Universal Robots PolyScope program: 2024dragon.urp

Program 2024dragon (installation=default directory=/programs createdIn=5.11.9.1010452 lastSavedIn=5.11.9.1010452 robotSerialNumber=20225200364)
Calibrated DH parameters: a=[0.00002, -0.569483, -0.54992, -0.00001, -0.000036, 0]; d=[0.180894, -146.691669, 192.918669, -46.053088, 0.119778, 0.115602]; alpha=[1.571425, -0.001534, 0.003359, 1.568739, -1.571477, 0]; deltaTheta=[0, 0.376258, -0.101074, -0.275185, -0.000002, 0]
Robot Program (runOnlyOnce=true)
  Script file /programs/usbdisk/new-robot/2024Dragon.script
    | def Machining1():
    |   # Default parameters:
    |   global speed_ms = 0.3
    |   global speed_rads = 0.75
    |   global accel_mss = 3
    |   global accel_radss = 1.2
    |   global blend_radius_m = 0.001
    | 
    |   # Add subprograms here
    |   # Start of main program
    |   # Program generated by RoboDK v5.6.5 for UR10e on 10/01/2024 16:23:47
    |   # Using nominal kinematics.
    |   blend_radius_m = 0.001
    |   speed_ms = 1.000
    |   # set_reference(p[0.335000, -0.152000, 0.002000, 0.000000, 0.000000, 0.000000])
    |   set_tcp(p[0.000000, 0.000000, 0.252000, 0.000000, 0.000000, 0.000000])
    |   # Show Tool
    |   movej([0.067194, -1.074636, -2.586948, -1.050805, 1.570796, 1.637990],accel_radss,speed_rads,0,blend_radius_m)
    |   movel([0.067194, -1.074636, -2.586948, -1.050805, 1.570796, 1.637990],accel_mss,speed_ms,0,blend_radius_m)
    |   # Splitting Linear movement in 32 (instruction 7: MoveL 3)
    |   movel([0.067194, -1.076085, -2.588243, -1.048061, 1.570796, 1.637990],accel_mss,speed_ms,0,blend_radius_m)
    |   movel([0.067194, -1.077544, -2.589536, -1.045309, 1.570796, 1.637990],accel_mss,speed_ms,0,blend_radius_m)
    |   movel([0.067194, -1.079013, -2.590827, -1.042549, 1.570796, 1.637990],accel_mss,speed_ms,0,blend_radius_m)
    |   movel([0.067194, -1.080492, -2.592116, -1.039781, 1.570796, 1.637990],accel_mss,speed_ms,0,blend_radius_m)
    |   movel([0.067194, -1.081981, -2.593403, -1.037005, 1.570796, 1.637990],accel_mss,speed_ms,0,blend_radius_m)
    |   movel([0.067194, -1.083480, -2.594688, -1.034221, 1.570796, 1.637990],accel_mss,speed_ms,0,blend_radius_m)
    |   movel([0.067194, -1.084989, -2.595971, -1.031429, 1.570796, 1.637990],accel_mss,speed_ms,0,blend_radius_m)
    |   movel([0.067194, -1.086509, -2.597251, -1.028629, 1.570796, 1.637990],accel_mss,speed_ms,0,blend_radius_m)
    |   movel([0.067194, -1.088039, -2.598529, -1.025821, 1.570796, 1.637990],accel_mss,speed_ms,0,blend_radius_m)
    |   movel([0.067194, -1.089579, -2.599806, -1.023004, 1.570796, 1.637990],accel_mss,speed_ms,0,blend_radius_m)
    |   movel([0.067194, -1.091130, -2.601080, -1.020179, 1.570796, 1.637990],accel_mss,speed_ms,0,blend_radius_m)
    |   movel([0.067194, -1.092691, -2.602351, -1.017346, 1.570796, 1.637990],accel_mss,speed_ms,0,blend_radius_m)
    |   movel([0.067194, -1.094263, -2.603621, -1.014505, 1.570796, 1.637990],accel_mss,speed_ms,0,blend_radius_m)
    |   movel([0.067194, -1.095846, -2.604888, -1.011655, 1.570796, 1.637990],accel_mss,speed_ms,0,blend_radius_m)
    |   movel([0.067194, -1.097439, -2.606154, -1.008797, 1.570796, 1.637990],accel_mss,speed_ms,0,blend_radius_m)
    |   movel([0.067194, -1.099042, -2.607417, -1.005930, 1.570796, 1.637990],accel_mss,speed_ms,0,blend_radius_m)
    |   movel([0.067194, -1.100657, -2.608677, -1.003055, 1.570796, 1.637990],accel_mss,speed_ms,0,blend_radius_m)
    |   movel([0.067194, -1.102282, -2.609936, -1.000171, 1.570796, 1.637990],accel_mss,speed_ms,0,blend_radius_m)
    |   movel([0.067194, -1.103918, -2.611192, -0.997279, 1.570796, 1.637990],accel_mss,speed_ms,0,blend_radius_m)
    |   movel([0.067194, -1.105565, -2.612446, -0.994378, 1.570796, 1.637990],accel_mss,speed_ms,0,blend_radius_m)
    |   movel([0.067194, -1.107223, -2.613698, -0.991469, 1.570796, 1.637990],accel_mss,speed_ms,0,blend_radius_m)
    |   movel([0.067194, -1.108891, -2.614947, -0.988551, 1.570796, 1.637990],accel_mss,speed_ms,0,blend_radius_m)
    |   movel([0.067194, -1.110571, -2.616194, -0.985624, 1.570796, 1.637990],accel_mss,speed_ms,0,blend_radius_m)
    |   movel([0.067194, -1.112262, -2.617439, -0.982688, 1.570796, 1.637990],accel_mss,speed_ms,0,blend_radius_m)
    |   movel([0.067194, -1.113964, -2.618681, -0.979744, 1.570796, 1.637990],accel_mss,speed_ms,0,blend_radius_m)
    |   movel([0.067194, -1.115677, -2.619921, -0.976791, 1.570796, 1.637990],accel_mss,speed_ms,0,blend_radius_m)
    |   movel([0.067194, -1.117402, -2.621159, -0.973829, 1.570796, 1.637990],accel_mss,speed_ms,0,blend_radius_m)
    |   movel([0.067194, -1.119137, -2.622394, -0.970858, 1.570796, 1.637990],accel_mss,speed_ms,0,blend_radius_m)
    |   movel([0.067194, -1.120884, -2.623627, -0.967878, 1.570796, 1.637990],accel_mss,speed_ms,0,blend_radius_m)
    |   movel([0.067194, -1.122643, -2.624857, -0.964889, 1.570796, 1.637990],accel_mss,speed_ms,0,blend_radius_m)
    |   movel([0.067194, -1.124413, -2.626085, -0.961891, 1.570796, 1.637990],accel_mss,speed_ms,0,blend_radius_m)
    |   movel([0.067194, -1.126194, -2.627311, -0.958884, 1.570796, 1.637990],accel_mss,speed_ms,0,blend_radius_m)
    |   movel([0.067194, -1.126194, -2.627311, -0.958884, 1.570796, 1.637990],accel_mss,speed_ms,0,blend_radius_m)
    |   speed_ms = 1.000
    |   movel([0.067194, -1.126194, -2.627311, -0.958884, 1.570796, 1.637990],accel_mss,speed_ms,0,blend_radius_m)
    |   movel([0.067194, -1.126194, -2.627311, -0.958884, 1.570796, 1.637990],accel_mss,speed_ms,0,blend_radius_m)
    |   movel([0.067194, -1.126194, -2.627311, -0.958884, 1.570796, 1.637990],accel_mss,speed_ms,0,blend_radius_m)
    |   speed_ms = 0.005
    |   # Splitting Linear movement in 22 (instruction 14: MoveL 8)
    |   movel([0.067194, -1.124466, -2.626123, -0.961800, 1.570796, 1.637990],accel_mss,speed_ms,0,blend_radius_m)
    |   movel([0.067194, -1.122750, -2.624932, -0.964708, 1.570796, 1.637990],accel_mss,speed_ms,0,blend_radius_m)
    |   movel([0.067194, -1.121044, -2.623739, -0.967606, 1.570796, 1.637990],accel_mss,speed_ms,0,blend_radius_m)
    |   movel([0.067194, -1.119348, -2.622544, -0.970497, 1.570796, 1.637990],accel_mss,speed_ms,0,blend_radius_m)
    |   movel([0.067194, -1.117664, -2.621346, -0.973379, 1.570796, 1.637990],accel_mss,speed_ms,0,blend_radius_m)
    |   movel([0.067194, -1.115990, -2.620146, -0.976253, 1.570796, 1.637990],accel_mss,speed_ms,0,blend_radius_m)
    |   movel([0.067194, -1.114326, -2.618944, -0.979118, 1.570796, 1.637990],accel_mss,speed_ms,0,blend_radius_m)
    |   movel([0.067194, -1.112674, -2.617740, -0.981975, 1.570796, 1.637990],accel_mss,speed_ms,0,blend_radius_m)
    |   movel([0.067194, -1.111031, -2.616534, -0.984824, 1.570796, 1.637990],accel_mss,speed_ms,0,blend_radius_m)
    |   movel([0.067194, -1.109399, -2.615325, -0.987665, 1.570796, 1.637990],accel_mss,speed_ms,0,blend_radius_m)
    |   movel([0.067194, -1.107778, -2.614114, -0.990497, 1.570796, 1.637990],accel_mss,speed_ms,0,blend_radius_m)
    |   movel([0.067194, -1.106166, -2.612901, -0.993321, 1.570796, 1.637990],accel_mss,speed_ms,0,blend_radius_m)
    |   movel([0.067194, -1.104565, -2.611686, -0.996137, 1.570796, 1.637990],accel_mss,speed_ms,0,blend_radius_m)
    |   movel([0.067194, -1.102975, -2.610469, -0.998945, 1.570796, 1.637990],accel_mss,speed_ms,0,blend_radius_m)
    |   movel([0.067194, -1.101394, -2.609250, -1.001745, 1.570796, 1.637990],accel_mss,speed_ms,0,blend_radius_m)
    |   movel([0.067194, -1.099824, -2.608028, -1.004537, 1.570796, 1.637990],accel_mss,speed_ms,0,blend_radius_m)
    |   movel([0.067194, -1.098263, -2.606805, -1.007321, 1.570796, 1.637990],accel_mss,speed_ms,0,blend_radius_m)
    |   movel([0.067194, -1.096713, -2.605579, -1.010097, 1.570796, 1.637990],accel_mss,speed_ms,0,blend_radius_m)
    |   movel([0.067194, -1.095173, -2.604351, -1.012865, 1.570796, 1.637990],accel_mss,speed_ms,0,blend_radius_m)
    |   movel([0.067194, -1.093643, -2.603121, -1.015625, 1.570796, 1.637990],accel_mss,speed_ms,0,blend_radius_m)
    |   movel([0.067194, -1.092123, -2.601889, -1.018377, 1.570796, 1.637990],accel_mss,speed_ms,0,blend_radius_m)
    |   movel([0.067194, -1.090612, -2.600655, -1.021122, 1.570796, 1.637990],accel_mss,speed_ms,0,blend_radius_m)
    |   speed_ms = 1.000
    |   # Splitting Linear movement in 22 (instruction 16: MoveL 9)
    |   movel([0.067194, -1.092123, -2.601889, -1.018377, 1.570796, 1.637990],accel_mss,speed_ms,0,blend_radius_m)
    |   movel([0.067194, -1.093643, -2.603121, -1.015625, 1.570796, 1.637990],accel_mss,speed_ms,0,blend_radius_m)
    |   movel([0.067194, -1.095173, -2.604351, -1.012865, 1.570796, 1.637990],accel_mss,speed_ms,0,blend_radius_m)
    |   movel([0.067194, -1.096713, -2.605579, -1.010097, 1.570796, 1.637990],accel_mss,speed_ms,0,blend_radius_m)
    |   movel([0.067194, -1.098263, -2.606805, -1.007321, 1.570796, 1.637990],accel_mss,speed_ms,0,blend_radius_m)
    |   movel([0.067194, -1.099824, -2.608028, -1.004537, 1.570796, 1.637990],accel_mss,speed_ms,0,blend_radius_m)
    |   movel([0.067194, -1.101394, -2.609250, -1.001745, 1.570796, 1.637990],accel_mss,speed_ms,0,blend_radius_m)
    |   movel([0.067194, -1.102975, -2.610469, -0.998945, 1.570796, 1.637990],accel_mss,speed_ms,0,blend_radius_m)
    |   movel([0.067194, -1.104565, -2.611686, -0.996137, 1.570796, 1.637990],accel_mss,speed_ms,0,blend_radius_m)
    |   movel([0.067194, -1.106166, -2.612901, -0.993321, 1.570796, 1.637990],accel_mss,speed_ms,0,blend_radius_m)
    |   movel([0.067194, -1.107778, -2.614114, -0.990497, 1.570796, 1.637990],accel_mss,speed_ms,0,blend_radius_m)
    |   movel([0.067194, -1.109399, -2.615325, -0.987665, 1.570796, 1.637990],accel_mss,speed_ms,0,blend_radius_m)
    |   movel([0.067194, -1.111031, -2.616534, -0.984824, 1.570796, 1.637990],accel_mss,speed_ms,0,blend_radius_m)
    |   movel([0.067194, -1.112674, -2.617740, -0.981975, 1.570796, 1.637990],accel_mss,speed_ms,0,blend_radius_m)
    |   movel([0.067194, -1.114326, -2.618944, -0.979118, 1.570796, 1.637990],accel_mss,speed_ms,0,blend_radius_m)
    |   movel([0.067194, -1.115990, -2.620146, -0.976253, 1.570796, 1.637990],accel_mss,speed_ms,0,blend_radius_m)
    |   movel([0.067194, -1.117664, -2.621346, -0.973379, 1.570796, 1.637990],accel_mss,speed_ms,0,blend_radius_m)
    |   movel([0.067194, -1.119348, -2.622544, -0.970497, 1.570796, 1.637990],accel_mss,speed_ms,0,blend_radius_m)
    |   movel([0.067194, -1.121044, -2.623739, -0.967606, 1.570796, 1.637990],accel_mss,speed_ms,0,blend_radius_m)
    |   movel([0.067194, -1.122750, -2.624932, -0.964708, 1.570796, 1.637990],accel_mss,speed_ms,0,blend_radius_m)
    |   movel([0.067194, -1.124466, -2.626123, -0.961800, 1.570796, 1.637990],accel_mss,speed_ms,0,blend_radius_m)
    |   movel([0.067194, -1.126194, -2.627311, -0.958884, 1.570796, 1.637990],accel_mss,speed_ms,0,blend_radius_m)
    |   speed_ms = 0.040
    |   movel([0.067194, -1.126194, -2.627311, -0.958884, 1.570796, 1.637990],accel_mss,speed_ms,0,blend_radius_m)
    |   speed_ms = 1.000
    |   movel([0.067194, -1.126194, -2.627311, -0.958884, 1.570796, 1.637990],accel_mss,speed_ms,0,blend_radius_m)
    |   # Splitting Linear movement in 38 (instruction 21: MoveL 12)
    |   movel([0.069828, -1.126252, -2.627286, -0.958852, 1.570796, 1.640625],accel_mss,speed_ms,0,blend_radius_m)
    |   movel([0.072458, -1.126317, -2.627257, -0.958815, 1.570796, 1.643255],accel_mss,speed_ms,0,blend_radius_m)
    |   movel([0.075084, -1.126391, -2.627225, -0.958773, 1.570796, 1.645881],accel_mss,speed_ms,0,blend_radius_m)
    |   movel([0.077706, -1.126473, -2.627189, -0.958727, 1.570796, 1.648503],accel_mss,speed_ms,0,blend_radius_m)
    |   movel([0.080324, -1.126562, -2.627150, -0.958677, 1.570796, 1.651120],accel_mss,speed_ms,0,blend_radius_m)
    |   movel([0.082938, -1.126660, -2.627107, -0.958622, 1.570796, 1.653734],accel_mss,speed_ms,0,blend_radius_m)
    |   movel([0.085547, -1.126766, -2.627061, -0.958562, 1.570796, 1.656343],accel_mss,speed_ms,0,blend_radius_m)
    |   movel([0.088152, -1.126880, -2.627011, -0.958498, 1.570796, 1.658948],accel_mss,speed_ms,0,blend_radius_m)
    |   movel([0.090752, -1.127001, -2.626958, -0.958430, 1.570796, 1.661549],accel_mss,speed_ms,0,blend_radius_m)
    |   movel([0.093349, -1.127131, -2.626901, -0.958357, 1.570796, 1.664145],accel_mss,speed_ms,0,blend_radius_m)
    |   movel([0.095940, -1.127269, -2.626841, -0.958279, 1.570796, 1.666737],accel_mss,speed_ms,0,blend_radius_m)
    |   movel([0.098528, -1.127415, -2.626777, -0.958197, 1.570796, 1.669324],accel_mss,speed_ms,0,blend_radius_m)
    |   movel([0.101111, -1.127568, -2.626710, -0.958111, 1.570796, 1.671907],accel_mss,speed_ms,0,blend_radius_m)
    |   movel([0.103689, -1.127730, -2.626639, -0.958020, 1.570796, 1.674485],accel_mss,speed_ms,0,blend_radius_m)
    |   movel([0.106263, -1.127899, -2.626565, -0.957925, 1.570796, 1.677059],accel_mss,speed_ms,0,blend_radius_m)
    |   movel([0.108832, -1.128077, -2.626487, -0.957825, 1.570796, 1.679629],accel_mss,speed_ms,0,blend_radius_m)
    |   movel([0.111397, -1.128262, -2.626406, -0.957721, 1.570796, 1.682193],accel_mss,speed_ms,0,blend_radius_m)
    |   movel([0.113957, -1.128456, -2.626321, -0.957612, 1.570796, 1.684754],accel_mss,speed_ms,0,blend_radius_m)
    |   movel([0.116513, -1.128657, -2.626233, -0.957499, 1.570796, 1.687309],accel_mss,speed_ms,0,blend_radius_m)
    |   movel([0.119064, -1.128866, -2.626141, -0.957382, 1.570796, 1.689860],accel_mss,speed_ms,0,blend_radius_m)
    |   movel([0.121610, -1.129083, -2.626045, -0.957260, 1.570796, 1.692406],accel_mss,speed_ms,0,blend_radius_m)
    |   movel([0.124151, -1.129308, -2.625947, -0.957134, 1.570796, 1.694947],accel_mss,speed_ms,0,blend_radius_m)
    |   movel([0.126687, -1.129541, -2.625844, -0.957004, 1.570796, 1.697484],accel_mss,speed_ms,0,blend_radius_m)
    |   movel([0.129219, -1.129781, -2.625738, -0.956869, 1.570796, 1.700016],accel_mss,speed_ms,0,blend_radius_m)
    |   movel([0.131746, -1.130030, -2.625629, -0.956730, 1.570796, 1.702542],accel_mss,speed_ms,0,blend_radius_m)
    |   movel([0.134268, -1.130286, -2.625516, -0.956587, 1.570796, 1.705065],accel_mss,speed_ms,0,blend_radius_m)
    |   movel([0.136785, -1.130550, -2.625400, -0.956439, 1.570796, 1.707582],accel_mss,speed_ms,0,blend_radius_m)
    |   movel([0.139298, -1.130822, -2.625280, -0.956287, 1.570796, 1.710094],accel_mss,speed_ms,0,blend_radius_m)
    |   movel([0.141805, -1.131102, -2.625156, -0.956131, 1.570796, 1.712601],accel_mss,speed_ms,0,blend_radius_m)
    |   movel([0.144307, -1.131389, -2.625030, -0.955970, 1.570796, 1.715104],accel_mss,speed_ms,0,blend_radius_m)
    |   movel([0.146805, -1.131684, -2.624899, -0.955805, 1.570796, 1.717601],accel_mss,speed_ms,0,blend_radius_m)
    |   movel([0.149297, -1.131987, -2.624765, -0.955636, 1.570796, 1.720093],accel_mss,speed_ms,0,blend_radius_m)
    |   movel([0.151784, -1.132298, -2.624628, -0.955463, 1.570796, 1.722581],accel_mss,speed_ms,0,blend_radius_m)
    |   movel([0.154267, -1.132616, -2.624487, -0.955286, 1.570796, 1.725063],accel_mss,speed_ms,0,blend_radius_m)
    |   movel([0.156744, -1.132942, -2.624343, -0.955104, 1.570796, 1.727540],accel_mss,speed_ms,0,blend_radius_m)
    |   movel([0.159216, -1.133276, -2.624195, -0.954918, 1.570796, 1.730012],accel_mss,speed_ms,0,blend_radius_m)
    |   movel([0.161683, -1.133617, -2.624043, -0.954728, 1.570796, 1.732479],accel_mss,speed_ms,0,blend_radius_m)
    |   movel([0.164144, -1.133966, -2.623888, -0.954534, 1.570796, 1.734941],accel_mss,speed_ms,0,blend_radius_m)
    |   speed_ms = 0.005
    |   # Splitting Linear movement in 22 (instruction 23: MoveL 13)
    |   movel([0.164144, -1.135705, -2.625067, -0.951617, 1.570796, 1.734941],accel_mss,speed_ms,0,blend_radius_m)
    |   movel([0.164144, -1.137454, -2.626244, -0.948691, 1.570796, 1.734941],accel_mss,speed_ms,0,blend_radius_m)
    |   movel([0.164144, -1.139214, -2.627418, -0.945757, 1.570796, 1.734941],accel_mss,speed_ms,0,blend_radius_m)
    |   movel([0.164144, -1.140985, -2.628590, -0.942814, 1.570796, 1.734941],accel_mss,speed_ms,0,blend_radius_m)
    |   movel([0.164144, -1.142767, -2.629760, -0.939862, 1.570796, 1.734941],accel_mss,speed_ms,0,blend_radius_m)
    |   movel([0.164144, -1.144560, -2.630927, -0.936902, 1.570796, 1.734941],accel_mss,speed_ms,0,blend_radius_m)
    |   movel([0.164144, -1.146364, -2.632091, -0.933934, 1.570796, 1.734941],accel_mss,speed_ms,0,blend_radius_m)
    |   movel([0.164144, -1.148179, -2.633254, -0.930957, 1.570796, 1.734941],accel_mss,speed_ms,0,blend_radius_m)
    |   movel([0.164144, -1.150005, -2.634414, -0.927971, 1.570796, 1.734941],accel_mss,speed_ms,0,blend_radius_m)
    |   movel([0.164144, -1.151842, -2.635571, -0.924976, 1.570796, 1.734941],accel_mss,speed_ms,0,blend_radius_m)
    |   movel([0.164144, -1.153690, -2.636726, -0.921973, 1.570796, 1.734941],accel_mss,speed_ms,0,blend_radius_m)
    |   movel([0.164144, -1.155550, -2.637879, -0.918961, 1.570796, 1.734941],accel_mss,speed_ms,0,blend_radius_m)
    |   movel([0.164144, -1.157420, -2.639029, -0.915940, 1.570796, 1.734941],accel_mss,speed_ms,0,blend_radius_m)
    |   movel([0.164144, -1.159302, -2.640176, -0.912911, 1.570796, 1.734941],accel_mss,speed_ms,0,blend_radius_m)
    |   movel([0.164144, -1.161196, -2.641321, -0.909872, 1.570796, 1.734941],accel_mss,speed_ms,0,blend_radius_m)
    |   movel([0.164144, -1.163101, -2.642463, -0.906825, 1.570796, 1.734941],accel_mss,speed_ms,0,blend_radius_m)
    |   movel([0.164144, -1.165017, -2.643603, -0.903769, 1.570796, 1.734941],accel_mss,speed_ms,0,blend_radius_m)
    |   movel([0.164144, -1.166945, -2.644741, -0.900704, 1.570796, 1.734941],accel_mss,speed_ms,0,blend_radius_m)
    |   movel([0.164144, -1.168884, -2.645876, -0.897629, 1.570796, 1.734941],accel_mss,speed_ms,0,blend_radius_m)
    |   movel([0.164144, -1.170835, -2.647008, -0.894546, 1.570796, 1.734941],accel_mss,speed_ms,0,blend_radius_m)
    |   movel([0.164144, -1.172797, -2.648137, -0.891454, 1.570796, 1.734941],accel_mss,speed_ms,0,blend_radius_m)
    |   movel([0.164144, -1.174772, -2.649264, -0.888353, 1.570796, 1.734941],accel_mss,speed_ms,0,blend_radius_m)
    |   speed_ms = 0.035
    |   movel([0.164993, -1.172613, -2.650270, -0.889506, 1.570796, 1.735790],accel_mss,speed_ms,0,blend_radius_m)
    |   movel([0.165155, -1.171113, -2.650966, -0.890310, 1.570796, 1.735952],accel_mss,speed_ms,0,blend_radius_m)
    |   movel([0.164874, -1.170165, -2.651404, -0.890819, 1.570796, 1.735671],accel_mss,speed_ms,0,blend_radius_m)
    |   movel([0.164399, -1.169671, -2.651633, -0.891085, 1.570796, 1.735195],accel_mss,speed_ms,0,blend_radius_m)
    |   movel([0.161880, -1.168870, -2.652002, -0.891517, 1.570796, 1.732676],accel_mss,speed_ms,0,blend_radius_m)
    |   movel([0.161427, -1.168227, -2.652299, -0.891864, 1.570796, 1.732224],accel_mss,speed_ms,0,blend_radius_m)
    |   movel([0.161378, -1.167640, -2.652568, -0.892180, 1.570796, 1.732174],accel_mss,speed_ms,0,blend_radius_m)
    |   movel([0.161619, -1.166900, -2.652908, -0.892581, 1.570796, 1.732416],accel_mss,speed_ms,0,blend_radius_m)
    |   movel([0.162186, -1.166146, -2.653254, -0.892989, 1.570796, 1.732982],accel_mss,speed_ms,0,blend_radius_m)
    |   movel([0.162955, -1.165553, -2.653526, -0.893311, 1.570796, 1.733751],accel_mss,speed_ms,0,blend_radius_m)
    |   movel([0.163842, -1.165169, -2.653701, -0.893519, 1.570796, 1.734638],accel_mss,speed_ms,0,blend_radius_m)
    |   movel([0.164754, -1.165038, -2.653761, -0.893590, 1.570796, 1.735550],accel_mss,speed_ms,0,blend_radius_m)
    |   movel([0.166318, -1.164944, -2.653804, -0.893641, 1.570796, 1.737114],accel_mss,speed_ms,0,blend_radius_m)
    |   movel([0.167392, -1.164661, -2.653933, -0.893795, 1.570796, 1.738188],accel_mss,speed_ms,0,blend_radius_m)
    |   movel([0.168112, -1.164264, -2.654114, -0.894010, 1.570796, 1.738908],accel_mss,speed_ms,0,blend_radius_m)
    |   movel([0.168622, -1.163824, -2.654315, -0.894250, 1.570796, 1.739418],accel_mss,speed_ms,0,blend_radius_m)
    |   movel([0.169089, -1.163137, -2.654628, -0.894624, 1.570796, 1.739886],accel_mss,speed_ms,0,blend_radius_m)
    |   movel([0.169480, -1.162013, -2.655138, -0.895237, 1.570796, 1.740276],accel_mss,speed_ms,0,blend_radius_m)
    |   movel([0.169481, -1.161424, -2.655406, -0.895560, 1.570796, 1.740277],accel_mss,speed_ms,0,blend_radius_m)
    |   movel([0.169274, -1.160885, -2.655650, -0.895854, 1.570796, 1.740071],accel_mss,speed_ms,0,blend_radius_m)
    |   movel([0.168785, -1.160454, -2.655845, -0.896090, 1.570796, 1.739581],accel_mss,speed_ms,0,blend_radius_m)
    |   movel([0.167958, -1.160181, -2.655968, -0.896240, 1.570796, 1.738755],accel_mss,speed_ms,0,blend_radius_m)
    |   speed_ms = 0.005
    |   # Splitting Linear movement in 6 (instruction 48: MoveL 36)
    |   movel([0.167958, -1.158728, -2.655131, -0.898529, 1.570796, 1.738755],accel_mss,speed_ms,0,blend_radius_m)
    |   movel([0.167958, -1.157282, -2.654293, -0.900814, 1.570796, 1.738755],accel_mss,speed_ms,0,blend_radius_m)
    |   movel([0.167958, -1.155842, -2.653454, -0.903093, 1.570796, 1.738755],accel_mss,speed_ms,0,blend_radius_m)
    |   movel([0.167958, -1.154408, -2.652613, -0.905368, 1.570796, 1.738755],accel_mss,speed_ms,0,blend_radius_m)
    |   movel([0.167958, -1.152981, -2.651771, -0.907637, 1.570796, 1.738755],accel_mss,speed_ms,0,blend_radius_m)
    |   movel([0.167958, -1.151560, -2.650928, -0.909901, 1.570796, 1.738755],accel_mss,speed_ms,0,blend_radius_m)
    |   speed_ms = 0.040
    |   # Splitting Linear movement in 4 (instruction 50: MoveL 37)
    |   movel([0.168272, -1.153369, -2.650117, -0.908903, 1.570796, 1.739068],accel_mss,speed_ms,0,blend_radius_m)
    |   movel([0.168584, -1.155175, -2.649304, -0.907909, 1.570796, 1.739381],accel_mss,speed_ms,0,blend_radius_m)
    |   movel([0.168895, -1.156978, -2.648490, -0.906921, 1.570796, 1.739692],accel_mss,speed_ms,0,blend_radius_m)
    |   movel([0.169205, -1.158777, -2.647674, -0.905937, 1.570796, 1.740001],accel_mss,speed_ms,0,blend_radius_m)
    |   speed_ms = 0.005
    |   # Splitting Linear movement in 6 (instruction 52: MoveL 38)
    |   movel([0.169205, -1.160197, -2.648513, -0.903680, 1.570796, 1.740001],accel_mss,speed_ms,0,blend_radius_m)
    |   movel([0.169205, -1.161622, -2.649350, -0.901417, 1.570796, 1.740001],accel_mss,speed_ms,0,blend_radius_m)
    |   movel([0.169205, -1.163054, -2.650186, -0.899149, 1.570796, 1.740001],accel_mss,speed_ms,0,blend_radius_m)
    |   movel([0.169205, -1.164492, -2.651020, -0.896877, 1.570796, 1.740001],accel_mss,speed_ms,0,blend_radius_m)
    |   movel([0.169205, -1.165937, -2.651853, -0.894599, 1.570796, 1.740001],accel_mss,speed_ms,0,blend_radius_m)
    |   movel([0.169205, -1.167388, -2.652684, -0.892317, 1.570796, 1.740001],accel_mss,speed_ms,0,blend_radius_m)
    |   speed_ms = 0.035
    |   movel([0.170114, -1.166953, -2.652884, -0.892552, 1.570796, 1.740910],accel_mss,speed_ms,0,blend_radius_m)
    |   movel([0.170952, -1.166789, -2.652959, -0.892641, 1.570796, 1.741748],accel_mss,speed_ms,0,blend_radius_m)
    |   movel([0.171650, -1.166893, -2.652911, -0.892584, 1.570796, 1.742446],accel_mss,speed_ms,0,blend_radius_m)
    |   movel([0.172147, -1.167265, -2.652741, -0.892383, 1.570796, 1.742943],accel_mss,speed_ms,0,blend_radius_m)
    |   movel([0.172364, -1.167756, -2.652515, -0.892118, 1.570796, 1.743160],accel_mss,speed_ms,0,blend_radius_m)
    |   movel([0.172398, -1.168357, -2.652239, -0.891793, 1.570796, 1.743194],accel_mss,speed_ms,0,blend_radius_m)
    |   movel([0.172257, -1.169008, -2.651939, -0.891442, 1.570796, 1.743053],accel_mss,speed_ms,0,blend_radius_m)
    |   movel([0.171937, -1.169655, -2.651640, -0.891094, 1.570796, 1.742733],accel_mss,speed_ms,0,blend_radius_m)
    |   movel([0.170592, -1.171154, -2.650947, -0.890288, 1.570796, 1.741389],accel_mss,speed_ms,0,blend_radius_m)
    |   movel([0.170274, -1.171690, -2.650699, -0.890001, 1.570796, 1.741070],accel_mss,speed_ms,0,blend_radius_m)
    |   movel([0.170191, -1.172226, -2.650450, -0.889713, 1.570796, 1.740988],accel_mss,speed_ms,0,blend_radius_m)
    |   movel([0.170379, -1.172720, -2.650220, -0.889449, 1.570796, 1.741175],accel_mss,speed_ms,0,blend_radius_m)
    |   movel([0.171372, -1.173703, -2.649763, -0.888923, 1.570796, 1.742169],accel_mss,speed_ms,0,blend_radius_m)
    |   movel([0.171436, -1.174467, -2.649406, -0.888515, 1.570796, 1.742232],accel_mss,speed_ms,0,blend_radius_m)
    |   movel([0.171020, -1.175716, -2.648823, -0.887850, 1.570796, 1.741816],accel_mss,speed_ms,0,blend_radius_m)
    |   movel([0.170183, -1.176926, -2.648256, -0.887207, 1.570796, 1.740979],accel_mss,speed_ms,0,blend_radius_m)
    |   movel([0.168973, -1.178188, -2.647663, -0.886538, 1.570796, 1.739769],accel_mss,speed_ms,0,blend_radius_m)
    |   movel([0.168429, -1.178790, -2.647379, -0.886220, 1.570796, 1.739226],accel_mss,speed_ms,0,blend_radius_m)
    |   movel([0.168360, -1.179147, -2.647211, -0.886031, 1.570796, 1.739156],accel_mss,speed_ms,0,blend_radius_m)
    |   movel([0.168489, -1.183287, -2.645249, -0.883852, 1.570796, 1.739286],accel_mss,speed_ms,0,blend_radius_m)
    |   movel([0.168759, -1.186160, -2.643878, -0.882351, 1.570796, 1.739555],accel_mss,speed_ms,0,blend_radius_m)
    |   movel([0.169225, -1.189338, -2.642350, -0.880701, 1.570796, 1.740022],accel_mss,speed_ms,0,blend_radius_m)
    |   movel([0.169930, -1.192649, -2.640747, -0.878993, 1.570796, 1.740726],accel_mss,speed_ms,0,blend_radius_m)
    |   movel([0.170917, -1.195924, -2.639150, -0.877315, 1.570796, 1.741713],accel_mss,speed_ms,0,blend_radius_m)
    |   movel([0.172230, -1.199002, -2.637638, -0.875749, 1.570796, 1.743026],accel_mss,speed_ms,0,blend_radius_m)
    |   movel([0.173910, -1.201718, -2.636295, -0.874376, 1.570796, 1.744706],accel_mss,speed_ms,0,blend_radius_m)
    |   speed_ms = 0.005
    |   # Splitting Linear movement in 6 (instruction 81: MoveL 65)
    |   movel([0.173910, -1.200279, -2.635489, -0.876622, 1.570796, 1.744706],accel_mss,speed_ms,0,blend_radius_m)
    |   movel([0.173910, -1.198846, -2.634680, -0.878863, 1.570796, 1.744706],accel_mss,speed_ms,0,blend_radius_m)
    |   movel([0.173910, -1.197418, -2.633871, -0.881100, 1.570796, 1.744706],accel_mss,speed_ms,0,blend_radius_m)
    |   movel([0.173910, -1.195997, -2.633060, -0.883332, 1.570796, 1.744706],accel_mss,speed_ms,0,blend_radius_m)
    |   movel([0.173910, -1.194582, -2.632247, -0.885560, 1.570796, 1.744706],accel_mss,speed_ms,0,blend_radius_m)
    |   movel([0.173910, -1.193172, -2.631433, -0.887784, 1.570796, 1.744706],accel_mss,speed_ms,0,blend_radius_m)
    |   speed_ms = 0.040
    |   # Splitting Linear movement in 8 (instruction 83: MoveL 66)
    |   movel([0.173598, -1.190744, -2.632621, -0.889025, 1.570796, 1.744395],accel_mss,speed_ms,0,blend_radius_m)
    |   movel([0.173285, -1.188308, -2.633805, -0.890275, 1.570796, 1.744081],accel_mss,speed_ms,0,blend_radius_m)
    |   movel([0.172970, -1.185866, -2.634987, -0.891536, 1.570796, 1.743766],accel_mss,speed_ms,0,blend_radius_m)
    |   movel([0.172653, -1.183417, -2.636165, -0.892806, 1.570796, 1.743449],accel_mss,speed_ms,0,blend_radius_m)
    |   movel([0.172334, -1.180962, -2.637341, -0.894087, 1.570796, 1.743130],accel_mss,speed_ms,0,blend_radius_m)
    |   movel([0.172013, -1.178499, -2.638513, -0.895377, 1.570796, 1.742810],accel_mss,speed_ms,0,blend_radius_m)
    |   movel([0.171691, -1.176030, -2.639682, -0.896677, 1.570796, 1.742487],accel_mss,speed_ms,0,blend_radius_m)
    |   movel([0.171366, -1.173553, -2.640848, -0.897987, 1.570796, 1.742163],accel_mss,speed_ms,0,blend_radius_m)
    |   speed_ms = 0.005
    |   # Splitting Linear movement in 6 (instruction 85: MoveL 67)
    |   movel([0.171366, -1.174969, -2.641676, -0.895744, 1.570796, 1.742163],accel_mss,speed_ms,0,blend_radius_m)
    |   movel([0.171366, -1.176391, -2.642503, -0.893495, 1.570796, 1.742163],accel_mss,speed_ms,0,blend_radius_m)
    |   movel([0.171366, -1.177819, -2.643328, -0.891242, 1.570796, 1.742163],accel_mss,speed_ms,0,blend_radius_m)
    |   movel([0.171366, -1.179253, -2.644152, -0.888984, 1.570796, 1.742163],accel_mss,speed_ms,0,blend_radius_m)
    |   movel([0.171366, -1.180693, -2.644974, -0.886722, 1.570796, 1.742163],accel_mss,speed_ms,0,blend_radius_m)
    |   movel([0.171366, -1.182140, -2.645795, -0.884454, 1.570796, 1.742163],accel_mss,speed_ms,0,blend_radius_m)
    |   speed_ms = 0.035
    |   movel([0.172318, -1.182599, -2.645577, -0.884213, 1.570796, 1.743114],accel_mss,speed_ms,0,blend_radius_m)
    |   movel([0.172755, -1.183182, -2.645299, -0.883907, 1.570796, 1.743551],accel_mss,speed_ms,0,blend_radius_m)
    |   movel([0.173064, -1.184692, -2.644580, -0.883117, 1.570796, 1.743861],accel_mss,speed_ms,0,blend_radius_m)
    |   movel([0.174344, -1.189035, -2.642496, -0.880858, 1.570796, 1.745141],accel_mss,speed_ms,0,blend_radius_m)
    |   movel([0.175391, -1.191364, -2.641371, -0.879655, 1.570796, 1.746188],accel_mss,speed_ms,0,blend_radius_m)
    |   speed_ms = 0.005
    |   # Splitting Linear movement in 4 (instruction 93: MoveL 73)
    |   movel([0.175391, -1.189201, -2.640149, -0.883039, 1.570796, 1.746188],accel_mss,speed_ms,0,blend_radius_m)
    |   movel([0.175391, -1.187052, -2.638923, -0.886413, 1.570796, 1.746188],accel_mss,speed_ms,0,blend_radius_m)
    |   movel([0.175391, -1.184917, -2.637695, -0.889777, 1.570796, 1.746188],accel_mss,speed_ms,0,blend_radius_m)
    |   movel([0.175391, -1.182795, -2.636464, -0.893130, 1.570796, 1.746188],accel_mss,speed_ms,0,blend_radius_m)
    |   speed_ms = 0.040
    |   # Splitting Linear movement in 6 (instruction 95: MoveL 74)
    |   movel([0.173869, -1.182309, -2.636697, -0.893384, 1.570796, 1.744666],accel_mss,speed_ms,0,blend_radius_m)
    |   movel([0.172344, -1.181825, -2.636928, -0.893636, 1.570796, 1.743141],accel_mss,speed_ms,0,blend_radius_m)
    |   movel([0.170816, -1.181344, -2.637158, -0.893887, 1.570796, 1.741613],accel_mss,speed_ms,0,blend_radius_m)
    |   movel([0.169286, -1.180866, -2.637386, -0.894136, 1.570796, 1.740082],accel_mss,speed_ms,0,blend_radius_m)
    |   movel([0.167752, -1.180392, -2.637612, -0.894385, 1.570796, 1.738548],accel_mss,speed_ms,0,blend_radius_m)
    |   movel([0.166215, -1.179921, -2.637837, -0.894631, 1.570796, 1.737012],accel_mss,speed_ms,0,blend_radius_m)
    |   speed_ms = 0.005
    |   # Splitting Linear movement in 4 (instruction 97: MoveL 75)
    |   movel([0.166215, -1.182044, -2.639072, -0.891274, 1.570796, 1.737012],accel_mss,speed_ms,0,blend_radius_m)
    |   movel([0.166215, -1.184180, -2.640303, -0.887906, 1.570796, 1.737012],accel_mss,speed_ms,0,blend_radius_m)
    |   movel([0.166215, -1.186331, -2.641531, -0.884527, 1.570796, 1.737012],accel_mss,speed_ms,0,blend_radius_m)
    |   movel([0.166215, -1.188495, -2.642756, -0.881138, 1.570796, 1.737012],accel_mss,speed_ms,0,blend_radius_m)
    |   speed_ms = 0.035
    |   movel([0.165570, -1.188509, -2.642749, -0.881130, 1.570796, 1.736366],accel_mss,speed_ms,0,blend_radius_m)
    |   movel([0.165117, -1.188390, -2.642807, -0.881192, 1.570796, 1.735913],accel_mss,speed_ms,0,blend_radius_m)
    |   movel([0.164703, -1.188087, -2.642953, -0.881350, 1.570796, 1.735500],accel_mss,speed_ms,0,blend_radius_m)
    |   movel([0.164445, -1.187572, -2.643200, -0.881617, 1.570796, 1.735241],accel_mss,speed_ms,0,blend_radius_m)
    |   movel([0.164378, -1.186989, -2.643480, -0.881920, 1.570796, 1.735174],accel_mss,speed_ms,0,blend_radius_m)
    |   movel([0.164545, -1.186209, -2.643854, -0.882326, 1.570796, 1.735341],accel_mss,speed_ms,0,blend_radius_m)
    |   movel([0.165033, -1.185319, -2.644280, -0.882790, 1.570796, 1.735829],accel_mss,speed_ms,0,blend_radius_m)
    |   movel([0.165777, -1.184484, -2.644679, -0.883226, 1.570796, 1.736573],accel_mss,speed_ms,0,blend_radius_m)
    |   movel([0.166708, -1.183776, -2.645017, -0.883597, 1.570796, 1.737504],accel_mss,speed_ms,0,blend_radius_m)
    |   movel([0.167760, -1.183265, -2.645260, -0.883864, 1.570796, 1.738556],accel_mss,speed_ms,0,blend_radius_m)
    |   speed_ms = 0.005
    |   # Splitting Linear movement in 4 (instruction 110: MoveL 86)
    |   movel([0.167760, -1.181099, -2.644029, -0.887261, 1.570796, 1.738556],accel_mss,speed_ms,0,blend_radius_m)
    |   movel([0.167760, -1.178946, -2.642795, -0.890648, 1.570796, 1.738556],accel_mss,speed_ms,0,blend_radius_m)
    |   movel([0.167760, -1.176806, -2.641558, -0.894024, 1.570796, 1.738556],accel_mss,speed_ms,0,blend_radius_m)
    |   movel([0.167760, -1.174681, -2.640318, -0.897390, 1.570796, 1.738556],accel_mss,speed_ms,0,blend_radius_m)
    |   speed_ms = 0.040
    |   # Splitting Linear movement in 4 (instruction 112: MoveL 87)
    |   movel([0.167066, -1.176975, -2.639235, -0.896179, 1.570796, 1.737863],accel_mss,speed_ms,0,blend_radius_m)
    |   movel([0.166376, -1.179262, -2.638151, -0.894977, 1.570796, 1.737173],accel_mss,speed_ms,0,blend_radius_m)
    |   movel([0.165689, -1.181540, -2.637064, -0.893784, 1.570796, 1.736486],accel_mss,speed_ms,0,blend_radius_m)
    |   movel([0.165006, -1.183811, -2.635976, -0.892602, 1.570796, 1.735802],accel_mss,speed_ms,0,blend_radius_m)
    |   speed_ms = 0.005
    |   # Splitting Linear movement in 4 (instruction 114: MoveL 88)
    |   movel([0.165006, -1.185932, -2.637207, -0.889250, 1.570796, 1.735802],accel_mss,speed_ms,0,blend_radius_m)
    |   movel([0.165006, -1.188067, -2.638434, -0.885888, 1.570796, 1.735802],accel_mss,speed_ms,0,blend_radius_m)
    |   movel([0.165006, -1.190215, -2.639658, -0.882516, 1.570796, 1.735802],accel_mss,speed_ms,0,blend_radius_m)
    |   movel([0.165006, -1.192377, -2.640879, -0.879133, 1.570796, 1.735802],accel_mss,speed_ms,0,blend_radius_m)
    |   speed_ms = 0.035
    |   movel([0.163332, -1.193015, -2.640569, -0.878805, 1.570796, 1.734128],accel_mss,speed_ms,0,blend_radius_m)
    |   movel([0.162063, -1.193271, -2.640445, -0.878674, 1.570796, 1.732859],accel_mss,speed_ms,0,blend_radius_m)
    |   movel([0.160779, -1.193238, -2.640460, -0.878690, 1.570796, 1.731575],accel_mss,speed_ms,0,blend_radius_m)
    |   movel([0.159860, -1.192671, -2.640736, -0.878982, 1.570796, 1.730656],accel_mss,speed_ms,0,blend_radius_m)
    |   movel([0.159365, -1.191925, -2.641098, -0.879365, 1.570796, 1.730161],accel_mss,speed_ms,0,blend_radius_m)
    |   movel([0.159176, -1.190790, -2.641649, -0.879951, 1.570796, 1.729972],accel_mss,speed_ms,0,blend_radius_m)
    |   movel([0.159392, -1.189814, -2.642120, -0.880455, 1.570796, 1.730188],accel_mss,speed_ms,0,blend_radius_m)
    |   movel([0.159907, -1.188849, -2.642586, -0.880954, 1.570796, 1.730703],accel_mss,speed_ms,0,blend_radius_m)
    |   movel([0.161408, -1.186486, -2.643722, -0.882182, 1.570796, 1.732204],accel_mss,speed_ms,0,blend_radius_m)
    |   movel([0.161780, -1.185616, -2.644138, -0.882635, 1.570796, 1.732576],accel_mss,speed_ms,0,blend_radius_m)
    |   movel([0.162148, -1.184263, -2.644784, -0.883341, 1.570796, 1.732944],accel_mss,speed_ms,0,blend_radius_m)
    |   movel([0.162268, -1.182733, -2.645513, -0.884143, 1.570796, 1.733064],accel_mss,speed_ms,0,blend_radius_m)
    |   movel([0.161896, -1.181326, -2.646181, -0.884882, 1.570796, 1.732692],accel_mss,speed_ms,0,blend_radius_m)
    |   movel([0.161088, -1.180451, -2.646595, -0.885343, 1.570796, 1.731884],accel_mss,speed_ms,0,blend_radius_m)
    |   movel([0.158772, -1.179531, -2.647030, -0.885828, 1.570796, 1.729569],accel_mss,speed_ms,0,blend_radius_m)
    |   movel([0.157403, -1.178904, -2.647325, -0.886159, 1.570796, 1.728199],accel_mss,speed_ms,0,blend_radius_m)
    |   movel([0.156927, -1.178484, -2.647523, -0.886381, 1.570796, 1.727723],accel_mss,speed_ms,0,blend_radius_m)
    |   movel([0.156681, -1.177962, -2.647769, -0.886658, 1.570796, 1.727477],accel_mss,speed_ms,0,blend_radius_m)
    |   movel([0.156623, -1.177403, -2.648032, -0.886954, 1.570796, 1.727419],accel_mss,speed_ms,0,blend_radius_m)
    |   movel([0.156725, -1.176861, -2.648286, -0.887242, 1.570796, 1.727521],accel_mss,speed_ms,0,blend_radius_m)
    |   movel([0.157215, -1.175937, -2.648719, -0.887733, 1.570796, 1.728011],accel_mss,speed_ms,0,blend_radius_m)
    |   movel([0.157906, -1.175147, -2.649089, -0.888153, 1.570796, 1.728703],accel_mss,speed_ms,0,blend_radius_m)
    |   movel([0.158997, -1.174248, -2.649509, -0.888632, 1.570796, 1.729793],accel_mss,speed_ms,0,blend_radius_m)
    |   speed_ms = 0.005
    |   # Splitting Linear movement in 4 (instruction 140: MoveL 112)
    |   movel([0.158997, -1.172077, -2.648268, -0.892044, 1.570796, 1.729793],accel_mss,speed_ms,0,blend_radius_m)
    |   movel([0.158997, -1.169919, -2.647025, -0.895445, 1.570796, 1.729793],accel_mss,speed_ms,0,blend_radius_m)
    |   movel([0.158997, -1.167776, -2.645778, -0.898834, 1.570796, 1.729793],accel_mss,speed_ms,0,blend_radius_m)
    |   movel([0.158997, -1.165647, -2.644528, -0.902213, 1.570796, 1.729793],accel_mss,speed_ms,0,blend_radius_m)
    |   speed_ms = 0.040
    |   # Splitting Linear movement in 8 (instruction 142: MoveL 113)
    |   movel([0.157361, -1.168361, -2.643273, -0.900756, 1.570796, 1.728157],accel_mss,speed_ms,0,blend_radius_m)
    |   movel([0.155733, -1.171063, -2.642014, -0.899311, 1.570796, 1.726530],accel_mss,speed_ms,0,blend_radius_m)
    |   movel([0.154115, -1.173755, -2.640754, -0.897881, 1.570796, 1.724911],accel_mss,speed_ms,0,blend_radius_m)
    |   movel([0.152505, -1.176435, -2.639490, -0.896463, 1.570796, 1.723301],accel_mss,speed_ms,0,blend_radius_m)
    |   movel([0.150903, -1.179105, -2.638225, -0.895059, 1.570796, 1.721699],accel_mss,speed_ms,0,blend_radius_m)
    |   movel([0.149309, -1.181764, -2.636957, -0.893667, 1.570796, 1.720106],accel_mss,speed_ms,0,blend_radius_m)
    |   movel([0.147724, -1.184413, -2.635687, -0.892289, 1.570796, 1.718521],accel_mss,speed_ms,0,blend_radius_m)
    |   movel([0.146148, -1.187050, -2.634415, -0.890924, 1.570796, 1.716944],accel_mss,speed_ms,0,blend_radius_m)
    |   speed_ms = 0.005
    |   # Splitting Linear movement in 6 (instruction 144: MoveL 114)
    |   movel([0.146148, -1.188462, -2.635233, -0.888694, 1.570796, 1.716944],accel_mss,speed_ms,0,blend_radius_m)
    |   movel([0.146148, -1.189880, -2.636050, -0.886459, 1.570796, 1.716944],accel_mss,speed_ms,0,blend_radius_m)
    |   movel([0.146148, -1.191303, -2.636865, -0.884220, 1.570796, 1.716944],accel_mss,speed_ms,0,blend_radius_m)
    |   movel([0.146148, -1.192733, -2.637679, -0.881977, 1.570796, 1.716944],accel_mss,speed_ms,0,blend_radius_m)
    |   movel([0.146148, -1.194168, -2.638492, -0.879729, 1.570796, 1.716944],accel_mss,speed_ms,0,blend_radius_m)
    |   movel([0.146148, -1.195610, -2.639303, -0.877476, 1.570796, 1.716944],accel_mss,speed_ms,0,blend_radius_m)
    |   speed_ms = 0.035
    |   movel([0.147576, -1.193096, -2.640530, -0.878764, 1.570796, 1.718372],accel_mss,speed_ms,0,blend_radius_m)
    |   movel([0.148654, -1.190486, -2.641795, -0.880107, 1.570796, 1.719450],accel_mss,speed_ms,0,blend_radius_m)
    |   movel([0.149343, -1.187857, -2.643063, -0.881469, 1.570796, 1.720139],accel_mss,speed_ms,0,blend_radius_m)
    |   movel([0.149605, -1.185292, -2.644293, -0.882804, 1.570796, 1.720402],accel_mss,speed_ms,0,blend_radius_m)
    |   movel([0.149400, -1.182861, -2.645452, -0.884076, 1.570796, 1.720197],accel_mss,speed_ms,0,blend_radius_m)
    |   movel([0.148686, -1.180651, -2.646500, -0.885237, 1.570796, 1.719482],accel_mss,speed_ms,0,blend_radius_m)
    |   movel([0.147429, -1.178738, -2.647404, -0.886247, 1.570796, 1.718225],accel_mss,speed_ms,0,blend_radius_m)
    |   movel([0.146580, -1.177922, -2.647788, -0.886679, 1.570796, 1.717376],accel_mss,speed_ms,0,blend_radius_m)
    |   movel([0.145581, -1.177214, -2.648121, -0.887055, 1.570796, 1.716378],accel_mss,speed_ms,0,blend_radius_m)
    |   movel([0.143703, -1.176382, -2.648511, -0.887496, 1.570796, 1.714499],accel_mss,speed_ms,0,blend_radius_m)
    |   movel([0.141523, -1.175958, -2.648709, -0.887721, 1.570796, 1.712319],accel_mss,speed_ms,0,blend_radius_m)
    |   movel([0.139094, -1.175946, -2.648715, -0.887728, 1.570796, 1.709891],accel_mss,speed_ms,0,blend_radius_m)
    |   movel([0.136483, -1.176341, -2.648530, -0.887518, 1.570796, 1.707280],accel_mss,speed_ms,0,blend_radius_m)
    |   movel([0.133748, -1.177140, -2.648155, -0.887094, 1.570796, 1.704544],accel_mss,speed_ms,0,blend_radius_m)
    |   movel([0.130956, -1.178336, -2.647593, -0.886460, 1.570796, 1.701752],accel_mss,speed_ms,0,blend_radius_m)
    |   movel([0.128168, -1.179925, -2.646844, -0.885620, 1.570796, 1.698964],accel_mss,speed_ms,0,blend_radius_m)
    |   movel([0.125445, -1.181900, -2.645909, -0.884580, 1.570796, 1.696242],accel_mss,speed_ms,0,blend_radius_m)
    |   movel([0.123177, -1.183926, -2.644945, -0.883518, 1.570796, 1.693973],accel_mss,speed_ms,0,blend_radius_m)
    |   movel([0.121158, -1.186091, -2.643911, -0.882387, 1.570796, 1.691954],accel_mss,speed_ms,0,blend_radius_m)
    |   movel([0.119398, -1.188357, -2.642823, -0.881209, 1.570796, 1.690194],accel_mss,speed_ms,0,blend_radius_m)
    |   movel([0.117907, -1.190684, -2.641699, -0.880005, 1.570796, 1.688703],accel_mss,speed_ms,0,blend_radius_m)
    |   movel([0.116702, -1.193026, -2.640563, -0.878799, 1.570796, 1.687498],accel_mss,speed_ms,0,blend_radius_m)
    |   movel([0.115785, -1.195347, -2.639432, -0.877610, 1.570796, 1.686581],accel_mss,speed_ms,0,blend_radius_m)
    |   movel([0.115164, -1.197608, -2.638324, -0.876457, 1.570796, 1.685961],accel_mss,speed_ms,0,blend_radius_m)
    |   movel([0.114855, -1.199769, -2.637259, -0.875360, 1.570796, 1.685651],accel_mss,speed_ms,0,blend_radius_m)
    |   movel([0.114871, -1.201943, -2.636184, -0.874262, 1.570796, 1.685667],accel_mss,speed_ms,0,blend_radius_m)
    |   movel([0.115242, -1.203901, -2.635210, -0.873277, 1.570796, 1.686039],accel_mss,speed_ms,0,blend_radius_m)
    |   movel([0.115949, -1.205627, -2.634349, -0.872413, 1.570796, 1.686746],accel_mss,speed_ms,0,blend_radius_m)
    |   movel([0.116970, -1.207102, -2.633610, -0.871677, 1.570796, 1.687767],accel_mss,speed_ms,0,blend_radius_m)
    |   movel([0.118284, -1.208309, -2.633004, -0.871076, 1.570796, 1.689080],accel_mss,speed_ms,0,blend_radius_m)
    |   movel([0.119877, -1.209228, -2.632541, -0.870620, 1.570796, 1.690673],accel_mss,speed_ms,0,blend_radius_m)
    |   movel([0.121731, -1.209843, -2.632231, -0.870315, 1.570796, 1.692527],accel_mss,speed_ms,0,blend_radius_m)
    |   movel([0.123825, -1.210135, -2.632084, -0.870170, 1.570796, 1.694621],accel_mss,speed_ms,0,blend_radius_m)
    |   speed_ms = 0.005
    |   # Splitting Linear movement in 6 (instruction 180: MoveL 148)
    |   movel([0.123825, -1.208700, -2.631283, -0.872407, 1.570796, 1.694621],accel_mss,speed_ms,0,blend_radius_m)
    |   movel([0.123825, -1.207270, -2.630481, -0.874638, 1.570796, 1.694621],accel_mss,speed_ms,0,blend_radius_m)
    |   movel([0.123825, -1.205846, -2.629677, -0.876866, 1.570796, 1.694621],accel_mss,speed_ms,0,blend_radius_m)
    |   movel([0.123825, -1.204428, -2.628872, -0.879089, 1.570796, 1.694621],accel_mss,speed_ms,0,blend_radius_m)
    |   movel([0.123825, -1.203016, -2.628065, -0.881307, 1.570796, 1.694621],accel_mss,speed_ms,0,blend_radius_m)
    |   movel([0.123825, -1.201610, -2.627258, -0.883522, 1.570796, 1.694621],accel_mss,speed_ms,0,blend_radius_m)
    |   speed_ms = 0.040
    |   # Splitting Linear movement in 6 (instruction 182: MoveL 149)
    |   movel([0.123400, -1.204254, -2.625933, -0.882202, 1.570796, 1.694196],accel_mss,speed_ms,0,blend_radius_m)
    |   movel([0.122977, -1.206888, -2.624606, -0.880895, 1.570796, 1.693773],accel_mss,speed_ms,0,blend_radius_m)
    |   movel([0.122557, -1.209512, -2.623277, -0.879600, 1.570796, 1.693353],accel_mss,speed_ms,0,blend_radius_m)
    |   movel([0.122139, -1.212127, -2.621945, -0.878318, 1.570796, 1.692935],accel_mss,speed_ms,0,blend_radius_m)
    |   movel([0.121723, -1.214731, -2.620610, -0.877048, 1.570796, 1.692520],accel_mss,speed_ms,0,blend_radius_m)
    |   movel([0.121310, -1.217326, -2.619273, -0.875790, 1.570796, 1.692107],accel_mss,speed_ms,0,blend_radius_m)
    |   speed_ms = 0.005
    |   # Splitting Linear movement in 4 (instruction 184: MoveL 150)
    |   movel([0.121310, -1.219428, -2.620467, -0.872494, 1.570796, 1.692107],accel_mss,speed_ms,0,blend_radius_m)
    |   movel([0.121310, -1.221542, -2.621658, -0.869188, 1.570796, 1.692107],accel_mss,speed_ms,0,blend_radius_m)
    |   movel([0.121310, -1.223669, -2.622846, -0.865873, 1.570796, 1.692107],accel_mss,speed_ms,0,blend_radius_m)
    |   movel([0.121310, -1.225809, -2.624031, -0.862549, 1.570796, 1.692107],accel_mss,speed_ms,0,blend_radius_m)
    |   speed_ms = 0.035
    |   movel([0.120799, -1.227627, -2.623079, -0.861683, 1.570796, 1.691596],accel_mss,speed_ms,0,blend_radius_m)
    |   movel([0.120802, -1.229138, -2.622285, -0.860966, 1.570796, 1.691599],accel_mss,speed_ms,0,blend_radius_m)
    |   movel([0.121019, -1.229913, -2.621877, -0.860599, 1.570796, 1.691816],accel_mss,speed_ms,0,blend_radius_m)
    |   movel([0.121434, -1.230653, -2.621486, -0.860250, 1.570796, 1.692230],accel_mss,speed_ms,0,blend_radius_m)
    |   movel([0.121889, -1.231103, -2.621248, -0.860037, 1.570796, 1.692685],accel_mss,speed_ms,0,blend_radius_m)
    |   movel([0.122486, -1.231439, -2.621071, -0.859879, 1.570796, 1.693283],accel_mss,speed_ms,0,blend_radius_m)
    |   movel([0.124000, -1.231773, -2.620894, -0.859722, 1.570796, 1.694796],accel_mss,speed_ms,0,blend_radius_m)
    |   movel([0.125766, -1.231652, -2.620958, -0.859779, 1.570796, 1.696563],accel_mss,speed_ms,0,blend_radius_m)
    |   movel([0.127575, -1.231068, -2.621267, -0.860054, 1.570796, 1.698371],accel_mss,speed_ms,0,blend_radius_m)
    |   movel([0.128818, -1.230382, -2.621629, -0.860377, 1.570796, 1.699614],accel_mss,speed_ms,0,blend_radius_m)
    |   movel([0.130001, -1.229510, -2.622089, -0.860790, 1.570796, 1.700797],accel_mss,speed_ms,0,blend_radius_m)
    |   movel([0.131092, -1.228491, -2.622625, -0.861273, 1.570796, 1.701888],accel_mss,speed_ms,0,blend_radius_m)
    |   movel([0.132063, -1.227358, -2.623220, -0.861811, 1.570796, 1.702859],accel_mss,speed_ms,0,blend_radius_m)
    |   movel([0.132877, -1.226151, -2.623852, -0.862386, 1.570796, 1.703673],accel_mss,speed_ms,0,blend_radius_m)
    |   movel([0.133501, -1.224904, -2.624504, -0.862982, 1.570796, 1.704298],accel_mss,speed_ms,0,blend_radius_m)
    |   movel([0.133904, -1.223655, -2.625154, -0.863580, 1.570796, 1.704700],accel_mss,speed_ms,0,blend_radius_m)
    |   movel([0.134047, -1.222444, -2.625783, -0.864162, 1.570796, 1.704843],accel_mss,speed_ms,0,blend_radius_m)
    |   movel([0.133954, -1.221539, -2.626252, -0.864598, 1.570796, 1.704750],accel_mss,speed_ms,0,blend_radius_m)
    |   movel([0.133682, -1.220746, -2.626662, -0.864981, 1.570796, 1.704479],accel_mss,speed_ms,0,blend_radius_m)
    |   movel([0.133244, -1.220078, -2.627007, -0.865304, 1.570796, 1.704040],accel_mss,speed_ms,0,blend_radius_m)
    |   movel([0.132648, -1.219547, -2.627281, -0.865561, 1.570796, 1.703444],accel_mss,speed_ms,0,blend_radius_m)
    |   movel([0.131913, -1.219158, -2.627481, -0.865749, 1.570796, 1.702709],accel_mss,speed_ms,0,blend_radius_m)
    |   movel([0.131046, -1.218930, -2.627599, -0.865860, 1.570796, 1.701843],accel_mss,speed_ms,0,blend_radius_m)
    |   movel([0.130062, -1.218866, -2.627632, -0.865891, 1.570796, 1.700859],accel_mss,speed_ms,0,blend_radius_m)
    |   movel([0.128976, -1.218981, -2.627572, -0.865835, 1.570796, 1.699772],accel_mss,speed_ms,0,blend_radius_m)
    |   speed_ms = 0.005
    |   # Splitting Linear movement in 4 (instruction 212: MoveL 176)
    |   movel([0.128976, -1.216836, -2.626380, -0.869172, 1.570796, 1.699772],accel_mss,speed_ms,0,blend_radius_m)
    |   movel([0.128976, -1.214705, -2.625185, -0.872499, 1.570796, 1.699772],accel_mss,speed_ms,0,blend_radius_m)
    |   movel([0.128976, -1.212585, -2.623987, -0.875817, 1.570796, 1.699772],accel_mss,speed_ms,0,blend_radius_m)
    |   movel([0.128976, -1.210479, -2.622785, -0.879125, 1.570796, 1.699772],accel_mss,speed_ms,0,blend_radius_m)
    |   speed_ms = 0.040
    |   # Splitting Linear movement in 4 (instruction 214: MoveL 177)
    |   movel([0.129350, -1.208215, -2.623935, -0.880239, 1.570796, 1.700147],accel_mss,speed_ms,0,blend_radius_m)
    |   movel([0.129726, -1.205943, -2.625083, -0.881363, 1.570796, 1.700523],accel_mss,speed_ms,0,blend_radius_m)
    |   movel([0.130104, -1.203664, -2.626229, -0.882496, 1.570796, 1.700901],accel_mss,speed_ms,0,blend_radius_m)
    |   movel([0.130484, -1.201377, -2.627374, -0.883638, 1.570796, 1.701281],accel_mss,speed_ms,0,blend_radius_m)
    |   speed_ms = 0.005
    |   # Splitting Linear movement in 6 (instruction 216: MoveL 178)
    |   movel([0.130484, -1.202784, -2.628182, -0.881424, 1.570796, 1.701281],accel_mss,speed_ms,0,blend_radius_m)
    |   movel([0.130484, -1.204196, -2.628988, -0.879205, 1.570796, 1.701281],accel_mss,speed_ms,0,blend_radius_m)
    |   movel([0.130484, -1.205614, -2.629794, -0.876981, 1.570796, 1.701281],accel_mss,speed_ms,0,blend_radius_m)
    |   movel([0.130484, -1.207038, -2.630597, -0.874754, 1.570796, 1.701281],accel_mss,speed_ms,0,blend_radius_m)
    |   movel([0.130484, -1.208467, -2.631400, -0.872522, 1.570796, 1.701281],accel_mss,speed_ms,0,blend_radius_m)
    |   movel([0.130484, -1.209903, -2.632201, -0.870285, 1.570796, 1.701281],accel_mss,speed_ms,0,blend_radius_m)
    |   speed_ms = 0.035
    |   movel([0.132665, -1.209505, -2.632401, -0.870482, 1.570796, 1.703461],accel_mss,speed_ms,0,blend_radius_m)
    |   movel([0.134695, -1.209419, -2.632445, -0.870525, 1.570796, 1.705491],accel_mss,speed_ms,0,blend_radius_m)
    |   movel([0.136561, -1.209630, -2.632338, -0.870420, 1.570796, 1.707357],accel_mss,speed_ms,0,blend_radius_m)
    |   movel([0.138244, -1.210127, -2.632088, -0.870174, 1.570796, 1.709040],accel_mss,speed_ms,0,blend_radius_m)
    |   movel([0.139728, -1.210897, -2.631699, -0.869794, 1.570796, 1.710524],accel_mss,speed_ms,0,blend_radius_m)
    |   movel([0.140999, -1.211919, -2.631181, -0.869289, 1.570796, 1.711795],accel_mss,speed_ms,0,blend_radius_m)
    |   movel([0.142039, -1.213181, -2.630540, -0.868668, 1.570796, 1.712836],accel_mss,speed_ms,0,blend_radius_m)
    |   movel([0.142838, -1.214670, -2.629782, -0.867937, 1.570796, 1.713634],accel_mss,speed_ms,0,blend_radius_m)
    |   movel([0.143240, -1.215895, -2.629156, -0.867338, 1.570796, 1.714036],accel_mss,speed_ms,0,blend_radius_m)
    |   movel([0.143450, -1.217164, -2.628506, -0.866718, 1.570796, 1.714246],accel_mss,speed_ms,0,blend_radius_m)
    |   movel([0.143494, -1.218458, -2.627842, -0.866089, 1.570796, 1.714290],accel_mss,speed_ms,0,blend_radius_m)
    |   movel([0.143387, -1.219764, -2.627169, -0.865456, 1.570796, 1.714184],accel_mss,speed_ms,0,blend_radius_m)
    |   movel([0.142831, -1.222338, -2.625838, -0.864213, 1.570796, 1.713627],accel_mss,speed_ms,0,blend_radius_m)
    |   movel([0.141958, -1.224755, -2.624581, -0.863053, 1.570796, 1.712754],accel_mss,speed_ms,0,blend_radius_m)
    |   movel([0.140945, -1.226894, -2.623463, -0.862032, 1.570796, 1.711741],accel_mss,speed_ms,0,blend_radius_m)
    |   movel([0.139971, -1.228624, -2.622555, -0.861209, 1.570796, 1.710767],accel_mss,speed_ms,0,blend_radius_m)
    |   movel([0.138805, -1.230386, -2.621627, -0.860376, 1.570796, 1.709601],accel_mss,speed_ms,0,blend_radius_m)
    |   movel([0.137417, -1.232076, -2.620734, -0.859579, 1.570796, 1.708214],accel_mss,speed_ms,0,blend_radius_m)
    |   movel([0.136043, -1.233556, -2.619948, -0.858885, 1.570796, 1.706840],accel_mss,speed_ms,0,blend_radius_m)
    |   movel([0.134255, -1.235249, -2.619047, -0.858093, 1.570796, 1.705052],accel_mss,speed_ms,0,blend_radius_m)
    |   movel([0.132090, -1.237000, -2.618112, -0.857278, 1.570796, 1.702886],accel_mss,speed_ms,0,blend_radius_m)
    |   movel([0.129574, -1.238659, -2.617222, -0.856508, 1.570796, 1.700370],accel_mss,speed_ms,0,blend_radius_m)
    |   movel([0.128192, -1.239407, -2.616820, -0.856163, 1.570796, 1.698989],accel_mss,speed_ms,0,blend_radius_m)
    |   movel([0.126735, -1.240072, -2.616461, -0.855855, 1.570796, 1.697531],accel_mss,speed_ms,0,blend_radius_m)
    |   movel([0.125203, -1.240642, -2.616154, -0.855593, 1.570796, 1.696000],accel_mss,speed_ms,0,blend_radius_m)
    |   movel([0.123602, -1.241094, -2.615910, -0.855385, 1.570796, 1.694399],accel_mss,speed_ms,0,blend_radius_m)
    |   movel([0.121219, -1.241502, -2.615689, -0.855197, 1.570796, 1.692016],accel_mss,speed_ms,0,blend_radius_m)
    |   movel([0.119139, -1.241573, -2.615651, -0.855165, 1.570796, 1.689935],accel_mss,speed_ms,0,blend_radius_m)
    |   movel([0.117360, -1.241384, -2.615753, -0.855252, 1.570796, 1.688156],accel_mss,speed_ms,0,blend_radius_m)
    |   movel([0.115877, -1.241020, -2.615950, -0.855419, 1.570796, 1.686673],accel_mss,speed_ms,0,blend_radius_m)
    |   movel([0.113778, -1.240076, -2.616459, -0.855854, 1.570796, 1.684574],accel_mss,speed_ms,0,blend_radius_m)
    |   movel([0.112821, -1.239374, -2.616837, -0.856178, 1.570796, 1.683617],accel_mss,speed_ms,0,blend_radius_m)
    |   movel([0.111813, -1.238211, -2.617462, -0.856716, 1.570796, 1.682609],accel_mss,speed_ms,0,blend_radius_m)
    |   movel([0.111054, -1.236855, -2.618189, -0.857345, 1.570796, 1.681850],accel_mss,speed_ms,0,blend_radius_m)
    |   movel([0.110545, -1.235333, -2.619002, -0.858054, 1.570796, 1.681342],accel_mss,speed_ms,0,blend_radius_m)
    |   movel([0.110292, -1.233669, -2.619889, -0.858832, 1.570796, 1.681089],accel_mss,speed_ms,0,blend_radius_m)
    |   movel([0.110292, -1.231885, -2.620835, -0.859669, 1.570796, 1.681089],accel_mss,speed_ms,0,blend_radius_m)
    |   movel([0.110550, -1.230005, -2.621828, -0.860556, 1.570796, 1.681346],accel_mss,speed_ms,0,blend_radius_m)
    |   movel([0.111063, -1.228059, -2.622852, -0.861478, 1.570796, 1.681859],accel_mss,speed_ms,0,blend_radius_m)
    |   movel([0.111838, -1.226070, -2.623894, -0.862424, 1.570796, 1.682635],accel_mss,speed_ms,0,blend_radius_m)
    |   movel([0.112974, -1.223883, -2.625035, -0.863471, 1.570796, 1.683770],accel_mss,speed_ms,0,blend_radius_m)
    |   movel([0.114216, -1.221973, -2.626027, -0.864389, 1.570796, 1.685013],accel_mss,speed_ms,0,blend_radius_m)
    |   movel([0.116502, -1.219141, -2.627490, -0.865758, 1.570796, 1.687299],accel_mss,speed_ms,0,blend_radius_m)
    |   speed_ms = 0.005
    |   # Splitting Linear movement in 4 (instruction 262: MoveL 222)
    |   movel([0.116502, -1.216996, -2.626298, -0.869094, 1.570796, 1.687299],accel_mss,speed_ms,0,blend_radius_m)
    |   movel([0.116502, -1.214865, -2.625103, -0.872421, 1.570796, 1.687299],accel_mss,speed_ms,0,blend_radius_m)
    |   movel([0.116502, -1.212746, -2.623905, -0.875739, 1.570796, 1.687299],accel_mss,speed_ms,0,blend_radius_m)
    |   movel([0.116502, -1.210639, -2.622703, -0.879046, 1.570796, 1.687299],accel_mss,speed_ms,0,blend_radius_m)
    |   speed_ms = 0.040
    |   # Splitting Linear movement in 8 (instruction 264: MoveL 223)
    |   movel([0.117942, -1.208307, -2.623888, -0.880194, 1.570796, 1.688738],accel_mss,speed_ms,0,blend_radius_m)
    |   movel([0.119388, -1.205967, -2.625071, -0.881351, 1.570796, 1.690184],accel_mss,speed_ms,0,blend_radius_m)
    |   movel([0.120840, -1.203618, -2.626253, -0.882519, 1.570796, 1.691637],accel_mss,speed_ms,0,blend_radius_m)
    |   movel([0.122300, -1.201260, -2.627432, -0.883697, 1.570796, 1.693096],accel_mss,speed_ms,0,blend_radius_m)
    |   movel([0.123766, -1.198895, -2.628609, -0.884885, 1.570796, 1.694562],accel_mss,speed_ms,0,blend_radius_m)
    |   movel([0.125239, -1.196521, -2.629785, -0.886083, 1.570796, 1.696035],accel_mss,speed_ms,0,blend_radius_m)
    |   movel([0.126719, -1.194138, -2.630959, -0.887292, 1.570796, 1.697515],accel_mss,speed_ms,0,blend_radius_m)
    |   movel([0.128206, -1.191747, -2.632131, -0.888511, 1.570796, 1.699002],accel_mss,speed_ms,0,blend_radius_m)
    |   speed_ms = 0.005
    |   # Splitting Linear movement in 4 (instruction 266: MoveL 224)
    |   movel([0.128206, -1.193864, -2.633353, -0.885172, 1.570796, 1.699002],accel_mss,speed_ms,0,blend_radius_m)
    |   movel([0.128206, -1.195995, -2.634571, -0.881823, 1.570796, 1.699002],accel_mss,speed_ms,0,blend_radius_m)
    |   movel([0.128206, -1.198139, -2.635787, -0.878463, 1.570796, 1.699002],accel_mss,speed_ms,0,blend_radius_m)
    |   movel([0.128206, -1.200296, -2.636999, -0.875094, 1.570796, 1.699002],accel_mss,speed_ms,0,blend_radius_m)
    |   speed_ms = 0.035
    |   movel([0.127187, -1.200028, -2.637132, -0.875229, 1.570796, 1.697983],accel_mss,speed_ms,0,blend_radius_m)
    |   movel([0.126349, -1.199560, -2.637362, -0.875466, 1.570796, 1.697145],accel_mss,speed_ms,0,blend_radius_m)
    |   movel([0.125697, -1.198914, -2.637681, -0.875794, 1.570796, 1.696493],accel_mss,speed_ms,0,blend_radius_m)
    |   movel([0.125240, -1.198107, -2.638078, -0.876203, 1.570796, 1.696036],accel_mss,speed_ms,0,blend_radius_m)
    |   movel([0.124981, -1.197166, -2.638541, -0.876682, 1.570796, 1.695777],accel_mss,speed_ms,0,blend_radius_m)
    |   movel([0.124927, -1.196106, -2.639061, -0.877223, 1.570796, 1.695723],accel_mss,speed_ms,0,blend_radius_m)
    |   movel([0.125080, -1.194952, -2.639625, -0.877812, 1.570796, 1.695876],accel_mss,speed_ms,0,blend_radius_m)
    |   movel([0.125453, -1.193722, -2.640225, -0.878442, 1.570796, 1.696249],accel_mss,speed_ms,0,blend_radius_m)
    |   movel([0.126069, -1.192439, -2.640849, -0.879101, 1.570796, 1.696865],accel_mss,speed_ms,0,blend_radius_m)
    |   movel([0.126889, -1.191204, -2.641448, -0.879737, 1.570796, 1.697686],accel_mss,speed_ms,0,blend_radius_m)
    |   movel([0.127869, -1.190046, -2.642008, -0.880335, 1.570796, 1.698665],accel_mss,speed_ms,0,blend_radius_m)
    |   movel([0.128970, -1.188985, -2.642520, -0.880884, 1.570796, 1.699767],accel_mss,speed_ms,0,blend_radius_m)
    |   movel([0.130144, -1.188047, -2.642972, -0.881370, 1.570796, 1.700941],accel_mss,speed_ms,0,blend_radius_m)
    |   movel([0.131351, -1.187249, -2.643356, -0.881785, 1.570796, 1.702148],accel_mss,speed_ms,0,blend_radius_m)
    |   movel([0.132544, -1.186624, -2.643655, -0.882110, 1.570796, 1.703340],accel_mss,speed_ms,0,blend_radius_m)
    |   movel([0.133685, -1.186185, -2.643866, -0.882338, 1.570796, 1.704481],accel_mss,speed_ms,0,blend_radius_m)
    |   movel([0.135141, -1.185914, -2.643995, -0.882479, 1.570796, 1.705937],accel_mss,speed_ms,0,blend_radius_m)
    |   movel([0.136561, -1.185982, -2.643963, -0.882444, 1.570796, 1.707358],accel_mss,speed_ms,0,blend_radius_m)
    |   movel([0.137825, -1.186412, -2.643757, -0.882220, 1.570796, 1.708621],accel_mss,speed_ms,0,blend_radius_m)
    |   movel([0.138822, -1.187213, -2.643373, -0.881803, 1.570796, 1.709618],accel_mss,speed_ms,0,blend_radius_m)
    |   movel([0.139429, -1.188408, -2.642798, -0.881183, 1.570796, 1.710225],accel_mss,speed_ms,0,blend_radius_m)
    |   movel([0.139535, -1.190006, -2.642028, -0.880356, 1.570796, 1.710331],accel_mss,speed_ms,0,blend_radius_m)
    |   movel([0.139367, -1.190961, -2.641566, -0.879862, 1.570796, 1.710163],accel_mss,speed_ms,0,blend_radius_m)
    |   movel([0.139030, -1.192021, -2.641052, -0.879316, 1.570796, 1.709827],accel_mss,speed_ms,0,blend_radius_m)
    |   movel([0.138512, -1.193191, -2.640483, -0.878715, 1.570796, 1.709308],accel_mss,speed_ms,0,blend_radius_m)
    |   movel([0.137802, -1.194465, -2.639863, -0.878061, 1.570796, 1.708598],accel_mss,speed_ms,0,blend_radius_m)
    |   speed_ms = 0.005
    |   # Splitting Linear movement in 4 (instruction 295: MoveL 251)
    |   movel([0.137802, -1.192304, -2.638644, -0.881441, 1.570796, 1.708598],accel_mss,speed_ms,0,blend_radius_m)
    |   movel([0.137802, -1.190157, -2.637422, -0.884810, 1.570796, 1.708598],accel_mss,speed_ms,0,blend_radius_m)
    |   movel([0.137802, -1.188023, -2.636197, -0.888168, 1.570796, 1.708598],accel_mss,speed_ms,0,blend_radius_m)
    |   movel([0.137802, -1.185903, -2.634969, -0.891517, 1.570796, 1.708598],accel_mss,speed_ms,0,blend_radius_m)
    |   speed_ms = 0.040
    |   movel([0.142596, -1.184943, -2.635432, -0.892014, 1.570796, 1.713393],accel_mss,speed_ms,0,blend_radius_m)
    |   speed_ms = 0.005
    |   # Splitting Linear movement in 6 (instruction 299: MoveL 253)
    |   movel([0.142596, -1.186355, -2.636252, -0.889782, 1.570796, 1.713393],accel_mss,speed_ms,0,blend_radius_m)
    |   movel([0.142596, -1.187774, -2.637070, -0.887545, 1.570796, 1.713393],accel_mss,speed_ms,0,blend_radius_m)
    |   movel([0.142596, -1.189198, -2.637887, -0.885304, 1.570796, 1.713393],accel_mss,speed_ms,0,blend_radius_m)
    |   movel([0.142596, -1.190628, -2.638703, -0.883058, 1.570796, 1.713393],accel_mss,speed_ms,0,blend_radius_m)
    |   movel([0.142596, -1.192065, -2.639517, -0.880807, 1.570796, 1.713393],accel_mss,speed_ms,0,blend_radius_m)
    |   movel([0.142596, -1.193507, -2.640329, -0.878552, 1.570796, 1.713393],accel_mss,speed_ms,0,blend_radius_m)
    |   speed_ms = 0.035
    |   movel([0.141839, -1.194858, -2.639671, -0.877860, 1.570796, 1.712635],accel_mss,speed_ms,0,blend_radius_m)
    |   movel([0.141229, -1.196207, -2.639011, -0.877171, 1.570796, 1.712026],accel_mss,speed_ms,0,blend_radius_m)
    |   movel([0.140437, -1.198851, -2.637712, -0.875826, 1.570796, 1.711233],accel_mss,speed_ms,0,blend_radius_m)
    |   movel([0.140244, -1.200131, -2.637081, -0.875177, 1.570796, 1.711040],accel_mss,speed_ms,0,blend_radius_m)
    |   movel([0.140178, -1.201366, -2.636470, -0.874553, 1.570796, 1.710974],accel_mss,speed_ms,0,blend_radius_m)
    |   movel([0.140405, -1.203682, -2.635319, -0.873387, 1.570796, 1.711202],accel_mss,speed_ms,0,blend_radius_m)
    |   movel([0.141081, -1.205727, -2.634299, -0.872363, 1.570796, 1.711877],accel_mss,speed_ms,0,blend_radius_m)
    |   movel([0.142164, -1.207433, -2.633444, -0.871512, 1.570796, 1.712961],accel_mss,speed_ms,0,blend_radius_m)
    |   movel([0.143617, -1.208726, -2.632794, -0.870869, 1.570796, 1.714413],accel_mss,speed_ms,0,blend_radius_m)
    |   movel([0.144470, -1.209198, -2.632556, -0.870634, 1.570796, 1.715267],accel_mss,speed_ms,0,blend_radius_m)
    |   movel([0.145401, -1.209541, -2.632383, -0.870465, 1.570796, 1.716197],accel_mss,speed_ms,0,blend_radius_m)
    |   movel([0.146595, -1.209782, -2.632262, -0.870345, 1.570796, 1.717392],accel_mss,speed_ms,0,blend_radius_m)
    |   movel([0.147881, -1.209857, -2.632224, -0.870308, 1.570796, 1.718678],accel_mss,speed_ms,0,blend_radius_m)
    |   movel([0.149245, -1.209768, -2.632269, -0.870352, 1.570796, 1.720042],accel_mss,speed_ms,0,blend_radius_m)
    |   movel([0.150667, -1.209523, -2.632392, -0.870473, 1.570796, 1.721463],accel_mss,speed_ms,0,blend_radius_m)
    |   movel([0.152141, -1.209129, -2.632591, -0.870669, 1.570796, 1.722937],accel_mss,speed_ms,0,blend_radius_m)
    |   movel([0.153647, -1.208592, -2.632862, -0.870936, 1.570796, 1.724443],accel_mss,speed_ms,0,blend_radius_m)
    |   movel([0.155169, -1.207913, -2.633203, -0.871273, 1.570796, 1.725965],accel_mss,speed_ms,0,blend_radius_m)
    |   movel([0.156701, -1.207100, -2.633611, -0.871678, 1.570796, 1.727498],accel_mss,speed_ms,0,blend_radius_m)
    |   movel([0.158221, -1.206159, -2.634083, -0.872147, 1.570796, 1.729017],accel_mss,speed_ms,0,blend_radius_m)
    |   movel([0.159718, -1.205090, -2.634617, -0.872682, 1.570796, 1.730514],accel_mss,speed_ms,0,blend_radius_m)
    |   movel([0.161179, -1.203904, -2.635209, -0.873276, 1.570796, 1.731975],accel_mss,speed_ms,0,blend_radius_m)
    |   movel([0.162586, -1.202601, -2.635857, -0.873931, 1.570796, 1.733382],accel_mss,speed_ms,0,blend_radius_m)
    |   movel([0.163926, -1.201188, -2.636558, -0.874643, 1.570796, 1.734722],accel_mss,speed_ms,0,blend_radius_m)
    |   movel([0.165185, -1.199668, -2.637309, -0.875412, 1.570796, 1.735981],accel_mss,speed_ms,0,blend_radius_m)
    |   movel([0.166348, -1.198048, -2.638108, -0.876234, 1.570796, 1.737144],accel_mss,speed_ms,0,blend_radius_m)
    |   movel([0.167398, -1.196330, -2.638951, -0.877108, 1.570796, 1.738194],accel_mss,speed_ms,0,blend_radius_m)
    |   speed_ms = 0.005
    |   # Splitting Linear movement in 4 (instruction 329: MoveL 281)
    |   movel([0.167398, -1.194171, -2.637734, -0.880484, 1.570796, 1.738194],accel_mss,speed_ms,0,blend_radius_m)
    |   movel([0.167398, -1.192024, -2.636514, -0.883850, 1.570796, 1.738194],accel_mss,speed_ms,0,blend_radius_m)
    |   movel([0.167398, -1.189892, -2.635291, -0.887206, 1.570796, 1.738194],accel_mss,speed_ms,0,blend_radius_m)
    |   movel([0.167398, -1.187772, -2.634065, -0.890551, 1.570796, 1.738194],accel_mss,speed_ms,0,blend_radius_m)
    |   speed_ms = 0.040
    |   # Splitting Linear movement in 8 (instruction 331: MoveL 282)
    |   movel([0.164905, -1.188471, -2.633727, -0.890192, 1.570796, 1.735701],accel_mss,speed_ms,0,blend_radius_m)
    |   movel([0.162412, -1.189174, -2.633385, -0.889830, 1.570796, 1.733208],accel_mss,speed_ms,0,blend_radius_m)
    |   movel([0.159920, -1.189881, -2.633041, -0.889467, 1.570796, 1.730716],accel_mss,speed_ms,0,blend_radius_m)
    |   movel([0.157429, -1.190592, -2.632694, -0.889102, 1.570796, 1.728225],accel_mss,speed_ms,0,blend_radius_m)
    |   movel([0.154939, -1.191309, -2.632345, -0.888735, 1.570796, 1.725735],accel_mss,speed_ms,0,blend_radius_m)
    |   movel([0.152449, -1.192029, -2.631993, -0.888367, 1.570796, 1.723246],accel_mss,speed_ms,0,blend_radius_m)
    |   movel([0.149961, -1.192754, -2.631638, -0.887997, 1.570796, 1.720757],accel_mss,speed_ms,0,blend_radius_m)
    |   movel([0.147473, -1.193483, -2.631281, -0.887625, 1.570796, 1.718270],accel_mss,speed_ms,0,blend_radius_m)
    |   speed_ms = 0.005
    |   # Splitting Linear movement in 6 (instruction 333: MoveL 283)
    |   movel([0.147473, -1.194892, -2.632095, -0.885402, 1.570796, 1.718270],accel_mss,speed_ms,0,blend_radius_m)
    |   movel([0.147473, -1.196307, -2.632907, -0.883175, 1.570796, 1.718270],accel_mss,speed_ms,0,blend_radius_m)
    |   movel([0.147473, -1.197729, -2.633718, -0.880943, 1.570796, 1.718270],accel_mss,speed_ms,0,blend_radius_m)
    |   movel([0.147473, -1.199156, -2.634527, -0.878706, 1.570796, 1.718270],accel_mss,speed_ms,0,blend_radius_m)
    |   movel([0.147473, -1.200589, -2.635335, -0.876465, 1.570796, 1.718270],accel_mss,speed_ms,0,blend_radius_m)
    |   movel([0.147473, -1.202028, -2.636142, -0.874220, 1.570796, 1.718270],accel_mss,speed_ms,0,blend_radius_m)
    |   speed_ms = 0.035
    |   movel([0.147938, -1.202430, -2.635942, -0.874017, 1.570796, 1.718735],accel_mss,speed_ms,0,blend_radius_m)
    |   movel([0.149207, -1.203073, -2.635623, -0.873694, 1.570796, 1.720003],accel_mss,speed_ms,0,blend_radius_m)
    |   movel([0.150144, -1.203291, -2.635514, -0.873584, 1.570796, 1.720941],accel_mss,speed_ms,0,blend_radius_m)
    |   movel([0.151283, -1.203343, -2.635488, -0.873558, 1.570796, 1.722079],accel_mss,speed_ms,0,blend_radius_m)
    |   movel([0.152624, -1.203151, -2.635584, -0.873654, 1.570796, 1.723421],accel_mss,speed_ms,0,blend_radius_m)
    |   movel([0.154176, -1.202631, -2.635842, -0.873916, 1.570796, 1.724972],accel_mss,speed_ms,0,blend_radius_m)
    |   movel([0.155533, -1.201946, -2.636182, -0.874261, 1.570796, 1.726329],accel_mss,speed_ms,0,blend_radius_m)
    |   movel([0.156748, -1.201141, -2.636581, -0.874667, 1.570796, 1.727544],accel_mss,speed_ms,0,blend_radius_m)
    |   movel([0.158706, -1.199416, -2.637434, -0.875539, 1.570796, 1.729502],accel_mss,speed_ms,0,blend_radius_m)
    |   movel([0.159999, -1.197915, -2.638173, -0.876301, 1.570796, 1.730795],accel_mss,speed_ms,0,blend_radius_m)
    |   movel([0.160567, -1.197119, -2.638564, -0.876706, 1.570796, 1.731363],accel_mss,speed_ms,0,blend_radius_m)
    |   speed_ms = 0.005
    |   # Splitting Linear movement in 6 (instruction 347: MoveL 295)
    |   movel([0.160567, -1.195678, -2.637754, -0.878957, 1.570796, 1.731363],accel_mss,speed_ms,0,blend_radius_m)
    |   movel([0.160567, -1.194243, -2.636942, -0.881204, 1.570796, 1.731363],accel_mss,speed_ms,0,blend_radius_m)
    |   movel([0.160567, -1.192814, -2.636129, -0.883446, 1.570796, 1.731363],accel_mss,speed_ms,0,blend_radius_m)
    |   movel([0.160567, -1.191391, -2.635315, -0.885683, 1.570796, 1.731363],accel_mss,speed_ms,0,blend_radius_m)
    |   movel([0.160567, -1.189974, -2.634499, -0.887916, 1.570796, 1.731363],accel_mss,speed_ms,0,blend_radius_m)
    |   movel([0.160567, -1.188563, -2.633682, -0.890144, 1.570796, 1.731363],accel_mss,speed_ms,0,blend_radius_m)
    |   speed_ms = 0.040
    |   # Splitting Linear movement in 6 (instruction 349: MoveL 296)
    |   movel([0.159178, -1.190624, -2.632679, -0.889086, 1.570796, 1.729975],accel_mss,speed_ms,0,blend_radius_m)
    |   movel([0.157795, -1.192679, -2.631675, -0.888035, 1.570796, 1.728591],accel_mss,speed_ms,0,blend_radius_m)
    |   movel([0.156418, -1.194728, -2.630669, -0.886992, 1.570796, 1.727214],accel_mss,speed_ms,0,blend_radius_m)
    |   movel([0.155045, -1.196770, -2.629662, -0.885957, 1.570796, 1.725842],accel_mss,speed_ms,0,blend_radius_m)
    |   movel([0.153679, -1.198807, -2.628653, -0.884929, 1.570796, 1.724475],accel_mss,speed_ms,0,blend_radius_m)
    |   movel([0.152317, -1.200837, -2.627643, -0.883909, 1.570796, 1.723114],accel_mss,speed_ms,0,blend_radius_m)
    |   speed_ms = 0.005
    |   # Splitting Linear movement in 6 (instruction 351: MoveL 297)
    |   movel([0.152317, -1.202244, -2.628452, -0.881694, 1.570796, 1.723114],accel_mss,speed_ms,0,blend_radius_m)
    |   movel([0.152317, -1.203656, -2.629259, -0.879474, 1.570796, 1.723114],accel_mss,speed_ms,0,blend_radius_m)
    |   movel([0.152317, -1.205074, -2.630064, -0.877250, 1.570796, 1.723114],accel_mss,speed_ms,0,blend_radius_m)
    |   movel([0.152317, -1.206498, -2.630869, -0.875022, 1.570796, 1.723114],accel_mss,speed_ms,0,blend_radius_m)
    |   movel([0.152317, -1.207928, -2.631671, -0.872789, 1.570796, 1.723114],accel_mss,speed_ms,0,blend_radius_m)
    |   movel([0.152317, -1.209364, -2.632473, -0.870552, 1.570796, 1.723114],accel_mss,speed_ms,0,blend_radius_m)
    |   speed_ms = 0.035
    |   movel([0.152335, -1.210185, -2.632058, -0.870146, 1.570796, 1.723131],accel_mss,speed_ms,0,blend_radius_m)
    |   movel([0.152177, -1.211018, -2.631637, -0.869734, 1.570796, 1.722973],accel_mss,speed_ms,0,blend_radius_m)
    |   movel([0.151867, -1.211835, -2.631223, -0.869330, 1.570796, 1.722664],accel_mss,speed_ms,0,blend_radius_m)
    |   movel([0.151435, -1.212615, -2.630828, -0.868946, 1.570796, 1.722231],accel_mss,speed_ms,0,blend_radius_m)
    |   movel([0.150907, -1.213328, -2.630465, -0.868595, 1.570796, 1.721703],accel_mss,speed_ms,0,blend_radius_m)
    |   movel([0.150312, -1.213949, -2.630149, -0.868291, 1.570796, 1.721108],accel_mss,speed_ms,0,blend_radius_m)
    |   movel([0.149673, -1.214454, -2.629892, -0.868043, 1.570796, 1.720470],accel_mss,speed_ms,0,blend_radius_m)
    |   movel([0.149019, -1.214818, -2.629706, -0.867865, 1.570796, 1.719816],accel_mss,speed_ms,0,blend_radius_m)
    |   movel([0.148108, -1.215059, -2.629583, -0.867747, 1.570796, 1.718904],accel_mss,speed_ms,0,blend_radius_m)
    |   movel([0.147257, -1.214989, -2.629619, -0.867781, 1.570796, 1.718053],accel_mss,speed_ms,0,blend_radius_m)
    |   movel([0.146531, -1.214628, -2.629803, -0.867958, 1.570796, 1.717327],accel_mss,speed_ms,0,blend_radius_m)
    |   movel([0.145990, -1.213993, -2.630127, -0.868269, 1.570796, 1.716787],accel_mss,speed_ms,0,blend_radius_m)
    |   speed_ms = 0.005
    |   # Splitting Linear movement in 4 (instruction 366: MoveL 310)
    |   movel([0.145990, -1.211845, -2.628929, -0.871615, 1.570796, 1.716787],accel_mss,speed_ms,0,blend_radius_m)
    |   movel([0.145990, -1.209710, -2.627729, -0.874951, 1.570796, 1.716787],accel_mss,speed_ms,0,blend_radius_m)
    |   movel([0.145990, -1.207587, -2.626525, -0.878277, 1.570796, 1.716787],accel_mss,speed_ms,0,blend_radius_m)
    |   movel([0.145990, -1.205478, -2.625317, -0.881594, 1.570796, 1.716787],accel_mss,speed_ms,0,blend_radius_m)
    |   speed_ms = 0.040
    |   # Splitting Linear movement in 4 (instruction 368: MoveL 311)
    |   movel([0.147845, -1.205837, -2.625136, -0.881415, 1.570796, 1.718641],accel_mss,speed_ms,0,blend_radius_m)
    |   movel([0.149696, -1.206201, -2.624953, -0.881235, 1.570796, 1.720492],accel_mss,speed_ms,0,blend_radius_m)
    |   movel([0.151544, -1.206569, -2.624767, -0.881053, 1.570796, 1.722340],accel_mss,speed_ms,0,blend_radius_m)
    |   movel([0.153388, -1.206942, -2.624579, -0.880868, 1.570796, 1.724184],accel_mss,speed_ms,0,blend_radius_m)
    |   speed_ms = 0.005
    |   # Splitting Linear movement in 4 (instruction 370: MoveL 312)
    |   movel([0.153388, -1.209050, -2.625785, -0.877554, 1.570796, 1.724184],accel_mss,speed_ms,0,blend_radius_m)
    |   movel([0.153388, -1.211171, -2.626987, -0.874230, 1.570796, 1.724184],accel_mss,speed_ms,0,blend_radius_m)
    |   movel([0.153388, -1.213306, -2.628186, -0.870897, 1.570796, 1.724184],accel_mss,speed_ms,0,blend_radius_m)
    |   movel([0.153388, -1.215453, -2.629382, -0.867554, 1.570796, 1.724184],accel_mss,speed_ms,0,blend_radius_m)
    |   speed_ms = 0.035
    |   movel([0.154156, -1.215333, -2.629444, -0.867613, 1.570796, 1.724952],accel_mss,speed_ms,0,blend_radius_m)
    |   movel([0.154866, -1.215045, -2.629590, -0.867753, 1.570796, 1.725662],accel_mss,speed_ms,0,blend_radius_m)
    |   movel([0.155788, -1.214446, -2.629896, -0.868047, 1.570796, 1.726584],accel_mss,speed_ms,0,blend_radius_m)
    |   movel([0.156555, -1.213660, -2.630297, -0.868433, 1.570796, 1.727352],accel_mss,speed_ms,0,blend_radius_m)
    |   movel([0.157079, -1.212911, -2.630677, -0.868800, 1.570796, 1.727875],accel_mss,speed_ms,0,blend_radius_m)
    |   movel([0.157397, -1.212210, -2.631033, -0.869146, 1.570796, 1.728194],accel_mss,speed_ms,0,blend_radius_m)
    |   movel([0.157546, -1.211572, -2.631357, -0.869460, 1.570796, 1.728342],accel_mss,speed_ms,0,blend_radius_m)
    |   movel([0.157496, -1.210519, -2.631889, -0.869980, 1.570796, 1.728292],accel_mss,speed_ms,0,blend_radius_m)
    |   movel([0.157250, -1.209838, -2.632233, -0.870317, 1.570796, 1.728046],accel_mss,speed_ms,0,blend_radius_m)
    |   movel([0.157001, -1.209173, -2.632569, -0.870647, 1.570796, 1.727798],accel_mss,speed_ms,0,blend_radius_m)
    |   movel([0.156991, -1.208627, -2.632844, -0.870918, 1.570796, 1.727788],accel_mss,speed_ms,0,blend_radius_m)
    |   movel([0.157391, -1.207625, -2.633348, -0.871416, 1.570796, 1.728188],accel_mss,speed_ms,0,blend_radius_m)
    |   movel([0.158045, -1.206680, -2.633822, -0.871887, 1.570796, 1.728841],accel_mss,speed_ms,0,blend_radius_m)
    |   movel([0.158975, -1.205817, -2.634254, -0.872318, 1.570796, 1.729772],accel_mss,speed_ms,0,blend_radius_m)
    |   movel([0.160042, -1.205149, -2.634588, -0.872652, 1.570796, 1.730838],accel_mss,speed_ms,0,blend_radius_m)
    |   movel([0.161106, -1.204794, -2.634765, -0.872830, 1.570796, 1.731903],accel_mss,speed_ms,0,blend_radius_m)
    |   movel([0.161707, -1.204768, -2.634778, -0.872843, 1.570796, 1.732504],accel_mss,speed_ms,0,blend_radius_m)
    |   movel([0.162256, -1.204885, -2.634720, -0.872784, 1.570796, 1.733053],accel_mss,speed_ms,0,blend_radius_m)
    |   movel([0.163082, -1.205517, -2.634404, -0.872468, 1.570796, 1.733879],accel_mss,speed_ms,0,blend_radius_m)
    |   movel([0.163298, -1.206020, -2.634152, -0.872217, 1.570796, 1.734095],accel_mss,speed_ms,0,blend_radius_m)
    |   movel([0.163348, -1.206638, -2.633843, -0.871908, 1.570796, 1.734144],accel_mss,speed_ms,0,blend_radius_m)
    |   movel([0.163199, -1.207363, -2.633479, -0.871547, 1.570796, 1.733996],accel_mss,speed_ms,0,blend_radius_m)
    |   movel([0.162824, -1.208189, -2.633064, -0.871136, 1.570796, 1.733620],accel_mss,speed_ms,0,blend_radius_m)
    |   speed_ms = 0.005
    |   # Splitting Linear movement in 6 (instruction 396: MoveL 336)
    |   movel([0.162824, -1.206753, -2.632262, -0.873374, 1.570796, 1.733620],accel_mss,speed_ms,0,blend_radius_m)
    |   movel([0.162824, -1.205323, -2.631458, -0.875608, 1.570796, 1.733620],accel_mss,speed_ms,0,blend_radius_m)
    |   movel([0.162824, -1.203898, -2.630653, -0.877838, 1.570796, 1.733620],accel_mss,speed_ms,0,blend_radius_m)
    |   movel([0.162824, -1.202479, -2.629847, -0.880063, 1.570796, 1.733620],accel_mss,speed_ms,0,blend_radius_m)
    |   movel([0.162824, -1.201066, -2.629039, -0.882284, 1.570796, 1.733620],accel_mss,speed_ms,0,blend_radius_m)
    |   movel([0.162824, -1.199659, -2.628230, -0.884500, 1.570796, 1.733620],accel_mss,speed_ms,0,blend_radius_m)
    |   speed_ms = 0.040
    |   # Splitting Linear movement in 18 (instruction 398: MoveL 337)
    |   movel([0.160979, -1.202399, -2.626863, -0.883127, 1.570796, 1.731775],accel_mss,speed_ms,0,blend_radius_m)
    |   movel([0.159143, -1.205127, -2.625494, -0.881768, 1.570796, 1.729939],accel_mss,speed_ms,0,blend_radius_m)
    |   movel([0.157317, -1.207845, -2.624122, -0.880422, 1.570796, 1.728113],accel_mss,speed_ms,0,blend_radius_m)
    |   movel([0.155500, -1.210552, -2.622748, -0.879089, 1.570796, 1.726297],accel_mss,speed_ms,0,blend_radius_m)
    |   movel([0.153694, -1.213247, -2.621371, -0.877771, 1.570796, 1.724490],accel_mss,speed_ms,0,blend_radius_m)
    |   movel([0.151896, -1.215932, -2.619992, -0.876465, 1.570796, 1.722693],accel_mss,speed_ms,0,blend_radius_m)
    |   movel([0.150108, -1.218607, -2.618610, -0.875172, 1.570796, 1.720905],accel_mss,speed_ms,0,blend_radius_m)
    |   movel([0.148330, -1.221271, -2.617226, -0.873893, 1.570796, 1.719126],accel_mss,speed_ms,0,blend_radius_m)
    |   movel([0.146560, -1.223924, -2.615839, -0.872626, 1.570796, 1.717357],accel_mss,speed_ms,0,blend_radius_m)
    |   movel([0.144800, -1.226567, -2.614450, -0.871373, 1.570796, 1.715596],accel_mss,speed_ms,0,blend_radius_m)
    |   movel([0.143049, -1.229199, -2.613058, -0.870132, 1.570796, 1.713845],accel_mss,speed_ms,0,blend_radius_m)
    |   movel([0.141307, -1.231822, -2.611664, -0.868903, 1.570796, 1.712103],accel_mss,speed_ms,0,blend_radius_m)
    |   movel([0.139574, -1.234434, -2.610268, -0.867688, 1.570796, 1.710370],accel_mss,speed_ms,0,blend_radius_m)
    |   movel([0.137850, -1.237036, -2.608869, -0.866484, 1.570796, 1.708646],accel_mss,speed_ms,0,blend_radius_m)
    |   movel([0.136135, -1.239628, -2.607468, -0.865293, 1.570796, 1.706931],accel_mss,speed_ms,0,blend_radius_m)
    |   movel([0.134428, -1.242210, -2.606064, -0.864115, 1.570796, 1.705225],accel_mss,speed_ms,0,blend_radius_m)
    |   movel([0.132730, -1.244782, -2.604658, -0.862948, 1.570796, 1.703527],accel_mss,speed_ms,0,blend_radius_m)
    |   movel([0.131041, -1.247345, -2.603250, -0.861794, 1.570796, 1.701838],accel_mss,speed_ms,0,blend_radius_m)
    |   speed_ms = 0.005
    |   # Splitting Linear movement in 6 (instruction 400: MoveL 338)
    |   movel([0.131041, -1.248729, -2.604025, -0.859634, 1.570796, 1.701838],accel_mss,speed_ms,0,blend_radius_m)
    |   movel([0.131041, -1.250119, -2.604799, -0.857471, 1.570796, 1.701838],accel_mss,speed_ms,0,blend_radius_m)
    |   movel([0.131041, -1.251514, -2.605571, -0.855303, 1.570796, 1.701838],accel_mss,speed_ms,0,blend_radius_m)
    |   movel([0.131041, -1.252915, -2.606342, -0.853132, 1.570796, 1.701838],accel_mss,speed_ms,0,blend_radius_m)
    |   movel([0.131041, -1.254321, -2.607111, -0.850957, 1.570796, 1.701838],accel_mss,speed_ms,0,blend_radius_m)
    |   movel([0.131041, -1.255732, -2.607879, -0.848778, 1.570796, 1.701838],accel_mss,speed_ms,0,blend_radius_m)
    |   speed_ms = 0.035
    |   movel([0.131215, -1.256892, -2.607232, -0.848265, 1.570796, 1.702012],accel_mss,speed_ms,0,blend_radius_m)
    |   movel([0.131722, -1.258552, -2.606302, -0.847534, 1.570796, 1.702519],accel_mss,speed_ms,0,blend_radius_m)
    |   movel([0.132755, -1.260324, -2.605307, -0.846758, 1.570796, 1.703551],accel_mss,speed_ms,0,blend_radius_m)
    |   movel([0.133528, -1.261129, -2.604854, -0.846406, 1.570796, 1.704324],accel_mss,speed_ms,0,blend_radius_m)
    |   movel([0.134502, -1.261818, -2.604465, -0.846106, 1.570796, 1.705299],accel_mss,speed_ms,0,blend_radius_m)
    |   movel([0.135616, -1.262259, -2.604216, -0.845914, 1.570796, 1.706413],accel_mss,speed_ms,0,blend_radius_m)
    |   movel([0.137753, -1.262646, -2.603997, -0.845745, 1.570796, 1.708549],accel_mss,speed_ms,0,blend_radius_m)
    |   movel([0.139170, -1.262683, -2.603976, -0.845729, 1.570796, 1.709966],accel_mss,speed_ms,0,blend_radius_m)
    |   movel([0.140803, -1.262541, -2.604057, -0.845791, 1.570796, 1.711599],accel_mss,speed_ms,0,blend_radius_m)
    |   movel([0.142644, -1.262161, -2.604272, -0.845956, 1.570796, 1.713441],accel_mss,speed_ms,0,blend_radius_m)
    |   movel([0.144678, -1.261492, -2.604650, -0.846248, 1.570796, 1.715475],accel_mss,speed_ms,0,blend_radius_m)
    |   movel([0.146049, -1.260879, -2.604995, -0.846515, 1.570796, 1.716845],accel_mss,speed_ms,0,blend_radius_m)
    |   movel([0.148639, -1.259405, -2.605824, -0.847160, 1.570796, 1.719436],accel_mss,speed_ms,0,blend_radius_m)
    |   movel([0.150208, -1.258304, -2.606442, -0.847643, 1.570796, 1.721005],accel_mss,speed_ms,0,blend_radius_m)
    |   movel([0.151868, -1.256938, -2.607206, -0.848245, 1.570796, 1.722665],accel_mss,speed_ms,0,blend_radius_m)
    |   movel([0.153542, -1.255290, -2.608125, -0.848974, 1.570796, 1.724338],accel_mss,speed_ms,0,blend_radius_m)
    |   movel([0.155158, -1.253342, -2.609207, -0.849840, 1.570796, 1.725954],accel_mss,speed_ms,0,blend_radius_m)
    |   movel([0.156393, -1.251493, -2.610230, -0.850665, 1.570796, 1.727190],accel_mss,speed_ms,0,blend_radius_m)
    |   movel([0.157389, -1.249618, -2.611264, -0.851507, 1.570796, 1.728185],accel_mss,speed_ms,0,blend_radius_m)
    |   movel([0.158136, -1.247749, -2.612290, -0.852350, 1.570796, 1.728932],accel_mss,speed_ms,0,blend_radius_m)
    |   movel([0.158630, -1.245912, -2.613294, -0.853183, 1.570796, 1.729426],accel_mss,speed_ms,0,blend_radius_m)
    |   movel([0.158865, -1.244140, -2.614259, -0.853990, 1.570796, 1.729661],accel_mss,speed_ms,0,blend_radius_m)
    |   movel([0.158831, -1.242466, -2.615168, -0.854755, 1.570796, 1.729627],accel_mss,speed_ms,0,blend_radius_m)
    |   movel([0.158523, -1.240923, -2.616003, -0.855464, 1.570796, 1.729320],accel_mss,speed_ms,0,blend_radius_m)
    |   movel([0.157936, -1.239539, -2.616748, -0.856101, 1.570796, 1.728733],accel_mss,speed_ms,0,blend_radius_m)
    |   movel([0.157093, -1.238381, -2.617371, -0.856637, 1.570796, 1.727889],accel_mss,speed_ms,0,blend_radius_m)
    |   movel([0.156091, -1.237511, -2.617838, -0.857040, 1.570796, 1.726887],accel_mss,speed_ms,0,blend_radius_m)
    |   movel([0.155000, -1.236890, -2.618170, -0.857329, 1.570796, 1.725796],accel_mss,speed_ms,0,blend_radius_m)
    |   movel([0.153883, -1.236477, -2.618391, -0.857521, 1.570796, 1.724679],accel_mss,speed_ms,0,blend_radius_m)
    |   movel([0.151845, -1.236117, -2.618584, -0.857688, 1.570796, 1.722641],accel_mss,speed_ms,0,blend_radius_m)
    |   movel([0.150519, -1.236090, -2.618598, -0.857701, 1.570796, 1.721316],accel_mss,speed_ms,0,blend_radius_m)
    |   speed_ms = 0.005
    |   # Splitting Linear movement in 4 (instruction 434: MoveL 370)
    |   movel([0.150519, -1.233958, -2.617425, -0.861006, 1.570796, 1.721316],accel_mss,speed_ms,0,blend_radius_m)
    |   movel([0.150519, -1.231839, -2.616248, -0.864302, 1.570796, 1.721316],accel_mss,speed_ms,0,blend_radius_m)
    |   movel([0.150519, -1.229732, -2.615068, -0.867589, 1.570796, 1.721316],accel_mss,speed_ms,0,blend_radius_m)
    |   movel([0.150519, -1.227638, -2.613885, -0.870867, 1.570796, 1.721316],accel_mss,speed_ms,0,blend_radius_m)
    |   speed_ms = 0.040
    |   # Splitting Linear movement in 4 (instruction 436: MoveL 371)
    |   movel([0.149950, -1.229249, -2.613032, -0.870108, 1.570796, 1.720747],accel_mss,speed_ms,0,blend_radius_m)
    |   movel([0.149383, -1.230856, -2.612178, -0.869355, 1.570796, 1.720179],accel_mss,speed_ms,0,blend_radius_m)
    |   movel([0.148818, -1.232459, -2.611324, -0.868606, 1.570796, 1.719614],accel_mss,speed_ms,0,blend_radius_m)
    |   movel([0.148255, -1.234058, -2.610469, -0.867862, 1.570796, 1.719051],accel_mss,speed_ms,0,blend_radius_m)
    |   speed_ms = 0.005
    |   # Splitting Linear movement in 4 (instruction 438: MoveL 372)
    |   movel([0.148255, -1.236148, -2.611645, -0.864596, 1.570796, 1.719051],accel_mss,speed_ms,0,blend_radius_m)
    |   movel([0.148255, -1.238250, -2.612818, -0.861321, 1.570796, 1.719051],accel_mss,speed_ms,0,blend_radius_m)
    |   movel([0.148255, -1.240364, -2.613988, -0.858037, 1.570796, 1.719051],accel_mss,speed_ms,0,blend_radius_m)
    |   movel([0.148255, -1.242490, -2.615155, -0.854744, 1.570796, 1.719051],accel_mss,speed_ms,0,blend_radius_m)
    |   speed_ms = 0.035
    |   movel([0.148831, -1.242633, -2.615077, -0.854678, 1.570796, 1.719628],accel_mss,speed_ms,0,blend_radius_m)
    |   movel([0.149732, -1.243045, -2.614854, -0.854490, 1.570796, 1.720528],accel_mss,speed_ms,0,blend_radius_m)
    |   movel([0.150630, -1.243869, -2.614407, -0.854113, 1.570796, 1.721426],accel_mss,speed_ms,0,blend_radius_m)
    |   movel([0.150974, -1.244478, -2.614076, -0.853835, 1.570796, 1.721771],accel_mss,speed_ms,0,blend_radius_m)
    |   movel([0.151201, -1.245239, -2.613661, -0.853488, 1.570796, 1.721997],accel_mss,speed_ms,0,blend_radius_m)
    |   movel([0.151266, -1.246072, -2.613207, -0.853110, 1.570796, 1.722062],accel_mss,speed_ms,0,blend_radius_m)
    |   movel([0.151182, -1.246972, -2.612715, -0.852702, 1.570796, 1.721978],accel_mss,speed_ms,0,blend_radius_m)
    |   movel([0.150952, -1.247921, -2.612196, -0.852272, 1.570796, 1.721749],accel_mss,speed_ms,0,blend_radius_m)
    |   movel([0.150579, -1.248893, -2.611662, -0.851834, 1.570796, 1.721376],accel_mss,speed_ms,0,blend_radius_m)
    |   movel([0.150068, -1.249873, -2.611124, -0.851393, 1.570796, 1.720864],accel_mss,speed_ms,0,blend_radius_m)
    |   movel([0.149420, -1.250834, -2.610594, -0.850961, 1.570796, 1.720217],accel_mss,speed_ms,0,blend_radius_m)
    |   movel([0.148643, -1.251757, -2.610085, -0.850547, 1.570796, 1.719439],accel_mss,speed_ms,0,blend_radius_m)
    |   movel([0.147736, -1.252624, -2.609605, -0.850160, 1.570796, 1.718532],accel_mss,speed_ms,0,blend_radius_m)
    |   movel([0.146538, -1.253519, -2.609109, -0.849761, 1.570796, 1.717334],accel_mss,speed_ms,0,blend_radius_m)
    |   movel([0.145382, -1.254161, -2.608753, -0.849475, 1.570796, 1.716179],accel_mss,speed_ms,0,blend_radius_m)
    |   movel([0.144300, -1.254594, -2.608512, -0.849283, 1.570796, 1.715096],accel_mss,speed_ms,0,blend_radius_m)
    |   movel([0.143329, -1.254856, -2.608367, -0.849167, 1.570796, 1.714125],accel_mss,speed_ms,0,blend_radius_m)
    |   movel([0.141847, -1.255033, -2.608268, -0.849088, 1.570796, 1.712643],accel_mss,speed_ms,0,blend_radius_m)
    |   movel([0.141215, -1.255011, -2.608280, -0.849098, 1.570796, 1.712012],accel_mss,speed_ms,0,blend_radius_m)
    |   speed_ms = 0.005
    |   # Splitting Linear movement in 6 (instruction 460: MoveL 392)
    |   movel([0.141215, -1.253600, -2.607512, -0.851277, 1.570796, 1.712012],accel_mss,speed_ms,0,blend_radius_m)
    |   movel([0.141215, -1.252193, -2.606742, -0.853453, 1.570796, 1.712012],accel_mss,speed_ms,0,blend_radius_m)
    |   movel([0.141215, -1.250793, -2.605971, -0.855625, 1.570796, 1.712012],accel_mss,speed_ms,0,blend_radius_m)
    |   movel([0.141215, -1.249397, -2.605198, -0.857794, 1.570796, 1.712012],accel_mss,speed_ms,0,blend_radius_m)
    |   movel([0.141215, -1.248007, -2.604424, -0.859958, 1.570796, 1.712012],accel_mss,speed_ms,0,blend_radius_m)
    |   movel([0.141215, -1.246622, -2.603648, -0.862119, 1.570796, 1.712012],accel_mss,speed_ms,0,blend_radius_m)
    |   speed_ms = 0.040
    |   movel([0.137114, -1.246679, -2.603617, -0.862093, 1.570796, 1.707910],accel_mss,speed_ms,0,blend_radius_m)
    |   speed_ms = 0.005
    |   # Splitting Linear movement in 6 (instruction 464: MoveL 394)
    |   movel([0.137114, -1.248064, -2.604393, -0.859933, 1.570796, 1.707910],accel_mss,speed_ms,0,blend_radius_m)
    |   movel([0.137114, -1.249454, -2.605167, -0.857768, 1.570796, 1.707910],accel_mss,speed_ms,0,blend_radius_m)
    |   movel([0.137114, -1.250850, -2.605939, -0.855600, 1.570796, 1.707910],accel_mss,speed_ms,0,blend_radius_m)
    |   movel([0.137114, -1.252251, -2.606711, -0.853428, 1.570796, 1.707910],accel_mss,speed_ms,0,blend_radius_m)
    |   movel([0.137114, -1.253657, -2.607480, -0.851252, 1.570796, 1.707910],accel_mss,speed_ms,0,blend_radius_m)
    |   movel([0.137114, -1.255068, -2.608248, -0.849072, 1.570796, 1.707910],accel_mss,speed_ms,0,blend_radius_m)
    |   speed_ms = 0.035
    |   movel([0.137992, -1.253542, -2.609096, -0.849750, 1.570796, 1.708789],accel_mss,speed_ms,0,blend_radius_m)
    |   movel([0.139146, -1.251110, -2.610442, -0.850837, 1.570796, 1.709942],accel_mss,speed_ms,0,blend_radius_m)
    |   movel([0.139678, -1.249644, -2.611249, -0.851495, 1.570796, 1.710475],accel_mss,speed_ms,0,blend_radius_m)
    |   movel([0.140102, -1.248064, -2.612117, -0.852208, 1.570796, 1.710898],accel_mss,speed_ms,0,blend_radius_m)
    |   movel([0.140358, -1.246402, -2.613027, -0.852960, 1.570796, 1.711155],accel_mss,speed_ms,0,blend_radius_m)
    |   movel([0.140387, -1.244698, -2.613956, -0.853735, 1.570796, 1.711183],accel_mss,speed_ms,0,blend_radius_m)
    |   movel([0.140173, -1.243214, -2.614763, -0.854413, 1.570796, 1.710969],accel_mss,speed_ms,0,blend_radius_m)
    |   movel([0.139772, -1.241952, -2.615446, -0.854991, 1.570796, 1.710568],accel_mss,speed_ms,0,blend_radius_m)
    |   movel([0.139232, -1.240903, -2.616013, -0.855473, 1.570796, 1.710029],accel_mss,speed_ms,0,blend_radius_m)
    |   movel([0.138609, -1.240045, -2.616476, -0.855868, 1.570796, 1.709405],accel_mss,speed_ms,0,blend_radius_m)
    |   movel([0.137320, -1.238832, -2.617129, -0.856428, 1.570796, 1.708117],accel_mss,speed_ms,0,blend_radius_m)
    |   movel([0.136338, -1.238176, -2.617481, -0.856732, 1.570796, 1.707134],accel_mss,speed_ms,0,blend_radius_m)
    |   speed_ms = 0.005
    |   # Splitting Linear movement in 6 (instruction 479: MoveL 407)
    |   movel([0.136338, -1.236755, -2.616701, -0.858934, 1.570796, 1.707134],accel_mss,speed_ms,0,blend_radius_m)
    |   movel([0.136338, -1.235339, -2.615919, -0.861131, 1.570796, 1.707134],accel_mss,speed_ms,0,blend_radius_m)
    |   movel([0.136338, -1.233929, -2.615135, -0.863325, 1.570796, 1.707134],accel_mss,speed_ms,0,blend_radius_m)
    |   movel([0.136338, -1.232524, -2.614350, -0.865515, 1.570796, 1.707134],accel_mss,speed_ms,0,blend_radius_m)
    |   movel([0.136338, -1.231124, -2.613564, -0.867701, 1.570796, 1.707134],accel_mss,speed_ms,0,blend_radius_m)
    |   movel([0.136338, -1.229730, -2.612776, -0.869882, 1.570796, 1.707134],accel_mss,speed_ms,0,blend_radius_m)
    |   speed_ms = 0.040
    |   # Splitting Linear movement in 10 (instruction 481: MoveL 408)
    |   movel([0.134715, -1.231830, -2.611660, -0.868900, 1.570796, 1.705511],accel_mss,speed_ms,0,blend_radius_m)
    |   movel([0.133098, -1.233923, -2.610541, -0.867925, 1.570796, 1.703894],accel_mss,speed_ms,0,blend_radius_m)
    |   movel([0.131488, -1.236009, -2.609422, -0.866958, 1.570796, 1.702284],accel_mss,speed_ms,0,blend_radius_m)
    |   movel([0.129884, -1.238090, -2.608300, -0.865999, 1.570796, 1.700680],accel_mss,speed_ms,0,blend_radius_m)
    |   movel([0.128286, -1.240164, -2.607177, -0.865048, 1.570796, 1.699083],accel_mss,speed_ms,0,blend_radius_m)
    |   movel([0.126695, -1.242233, -2.606052, -0.864104, 1.570796, 1.697492],accel_mss,speed_ms,0,blend_radius_m)
    |   movel([0.125111, -1.244295, -2.604925, -0.863169, 1.570796, 1.695907],accel_mss,speed_ms,0,blend_radius_m)
    |   movel([0.123532, -1.246351, -2.603797, -0.862241, 1.570796, 1.694328],accel_mss,speed_ms,0,blend_radius_m)
    |   movel([0.121960, -1.248402, -2.602667, -0.861320, 1.570796, 1.692756],accel_mss,speed_ms,0,blend_radius_m)
    |   movel([0.120394, -1.250446, -2.601536, -0.860407, 1.570796, 1.691190],accel_mss,speed_ms,0,blend_radius_m)
    |   speed_ms = 0.005
    |   # Splitting Linear movement in 4 (instruction 483: MoveL 409)
    |   movel([0.120394, -1.252522, -2.602695, -0.857172, 1.570796, 1.691190],accel_mss,speed_ms,0,blend_radius_m)
    |   movel([0.120394, -1.254610, -2.603850, -0.853929, 1.570796, 1.691190],accel_mss,speed_ms,0,blend_radius_m)
    |   movel([0.120394, -1.256710, -2.605003, -0.850676, 1.570796, 1.691190],accel_mss,speed_ms,0,blend_radius_m)
    |   movel([0.120394, -1.258822, -2.606151, -0.847416, 1.570796, 1.691190],accel_mss,speed_ms,0,blend_radius_m)
    |   speed_ms = 0.035
    |   movel([0.119725, -1.258727, -2.606204, -0.847457, 1.570796, 1.690521],accel_mss,speed_ms,0,blend_radius_m)
    |   movel([0.119088, -1.258483, -2.606341, -0.847565, 1.570796, 1.689884],accel_mss,speed_ms,0,blend_radius_m)
    |   movel([0.117994, -1.257616, -2.606827, -0.847946, 1.570796, 1.688790],accel_mss,speed_ms,0,blend_radius_m)
    |   movel([0.117260, -1.256365, -2.607526, -0.848498, 1.570796, 1.688056],accel_mss,speed_ms,0,blend_radius_m)
    |   movel([0.117072, -1.255639, -2.607931, -0.848819, 1.570796, 1.687868],accel_mss,speed_ms,0,blend_radius_m)
    |   movel([0.117032, -1.254873, -2.608357, -0.849159, 1.570796, 1.687829],accel_mss,speed_ms,0,blend_radius_m)
    |   movel([0.117218, -1.253699, -2.609009, -0.849681, 1.570796, 1.688015],accel_mss,speed_ms,0,blend_radius_m)
    |   movel([0.117620, -1.252583, -2.609628, -0.850178, 1.570796, 1.688417],accel_mss,speed_ms,0,blend_radius_m)
    |   movel([0.118170, -1.251550, -2.610199, -0.850640, 1.570796, 1.688966],accel_mss,speed_ms,0,blend_radius_m)
    |   movel([0.118809, -1.250616, -2.610714, -0.851059, 1.570796, 1.689605],accel_mss,speed_ms,0,blend_radius_m)
    |   movel([0.120091, -1.249147, -2.611523, -0.851719, 1.570796, 1.690887],accel_mss,speed_ms,0,blend_radius_m)
    |   movel([0.121848, -1.247644, -2.612347, -0.852398, 1.570796, 1.692644],accel_mss,speed_ms,0,blend_radius_m)
    |   movel([0.123196, -1.246809, -2.612805, -0.852776, 1.570796, 1.693992],accel_mss,speed_ms,0,blend_radius_m)
    |   movel([0.124904, -1.246111, -2.613186, -0.853092, 1.570796, 1.695700],accel_mss,speed_ms,0,blend_radius_m)
    |   movel([0.125863, -1.245904, -2.613299, -0.853187, 1.570796, 1.696660],accel_mss,speed_ms,0,blend_radius_m)
    |   movel([0.126879, -1.245832, -2.613338, -0.853219, 1.570796, 1.697675],accel_mss,speed_ms,0,blend_radius_m)
    |   movel([0.127900, -1.245949, -2.613274, -0.853166, 1.570796, 1.698696],accel_mss,speed_ms,0,blend_radius_m)
    |   movel([0.128817, -1.246275, -2.613096, -0.853018, 1.570796, 1.699613],accel_mss,speed_ms,0,blend_radius_m)
    |   movel([0.129588, -1.246808, -2.612805, -0.852776, 1.570796, 1.700384],accel_mss,speed_ms,0,blend_radius_m)
    |   movel([0.130186, -1.247536, -2.612407, -0.852446, 1.570796, 1.700982],accel_mss,speed_ms,0,blend_radius_m)
    |   movel([0.130572, -1.248457, -2.611902, -0.852030, 1.570796, 1.701368],accel_mss,speed_ms,0,blend_radius_m)
    |   movel([0.130718, -1.249561, -2.611295, -0.851533, 1.570796, 1.701514],accel_mss,speed_ms,0,blend_radius_m)
    |   movel([0.130588, -1.250841, -2.610590, -0.850958, 1.570796, 1.701385],accel_mss,speed_ms,0,blend_radius_m)
    |   movel([0.130148, -1.252291, -2.609789, -0.850309, 1.570796, 1.700944],accel_mss,speed_ms,0,blend_radius_m)
    |   speed_ms = 0.005
    |   # Splitting Linear movement in 6 (instruction 510: MoveL 434)
    |   movel([0.130148, -1.250878, -2.609019, -0.852492, 1.570796, 1.700944],accel_mss,speed_ms,0,blend_radius_m)
    |   movel([0.130148, -1.249470, -2.608247, -0.854672, 1.570796, 1.700944],accel_mss,speed_ms,0,blend_radius_m)
    |   movel([0.130148, -1.248067, -2.607474, -0.856847, 1.570796, 1.700944],accel_mss,speed_ms,0,blend_radius_m)
    |   movel([0.130148, -1.246670, -2.606700, -0.859019, 1.570796, 1.700944],accel_mss,speed_ms,0,blend_radius_m)
    |   movel([0.130148, -1.245278, -2.605923, -0.861187, 1.570796, 1.700944],accel_mss,speed_ms,0,blend_radius_m)
    |   movel([0.130148, -1.243892, -2.605146, -0.863351, 1.570796, 1.700944],accel_mss,speed_ms,0,blend_radius_m)
    |   speed_ms = 0.040
    |   # Splitting Linear movement in 20 (instruction 512: MoveL 435)
    |   movel([0.128701, -1.246423, -2.603758, -0.862208, 1.570796, 1.699497],accel_mss,speed_ms,0,blend_radius_m)
    |   movel([0.127261, -1.248943, -2.602368, -0.861078, 1.570796, 1.698058],accel_mss,speed_ms,0,blend_radius_m)
    |   movel([0.125829, -1.251455, -2.600976, -0.859958, 1.570796, 1.696625],accel_mss,speed_ms,0,blend_radius_m)
    |   movel([0.124404, -1.253957, -2.599582, -0.858851, 1.570796, 1.695200],accel_mss,speed_ms,0,blend_radius_m)
    |   movel([0.122986, -1.256449, -2.598185, -0.857755, 1.570796, 1.693783],accel_mss,speed_ms,0,blend_radius_m)
    |   movel([0.121576, -1.258932, -2.596787, -0.856670, 1.570796, 1.692372],accel_mss,speed_ms,0,blend_radius_m)
    |   movel([0.120172, -1.261406, -2.595387, -0.855597, 1.570796, 1.690968],accel_mss,speed_ms,0,blend_radius_m)
    |   movel([0.118776, -1.263871, -2.593984, -0.854534, 1.570796, 1.689572],accel_mss,speed_ms,0,blend_radius_m)
    |   movel([0.117386, -1.266326, -2.592580, -0.853483, 1.570796, 1.688183],accel_mss,speed_ms,0,blend_radius_m)
    |   movel([0.116004, -1.268772, -2.591173, -0.852443, 1.570796, 1.686800],accel_mss,speed_ms,0,blend_radius_m)
    |   movel([0.114628, -1.271210, -2.589765, -0.851415, 1.570796, 1.685424],accel_mss,speed_ms,0,blend_radius_m)
    |   movel([0.113259, -1.273638, -2.588354, -0.850396, 1.570796, 1.684056],accel_mss,speed_ms,0,blend_radius_m)
    |   movel([0.111897, -1.276058, -2.586942, -0.849389, 1.570796, 1.682694],accel_mss,speed_ms,0,blend_radius_m)
    |   movel([0.110542, -1.278469, -2.585527, -0.848393, 1.570796, 1.681338],accel_mss,speed_ms,0,blend_radius_m)
    |   movel([0.109193, -1.280871, -2.584111, -0.847407, 1.570796, 1.679990],accel_mss,speed_ms,0,blend_radius_m)
    |   movel([0.107851, -1.283265, -2.582693, -0.846432, 1.570796, 1.678648],accel_mss,speed_ms,0,blend_radius_m)
    |   movel([0.106516, -1.285650, -2.581273, -0.845467, 1.570796, 1.677312],accel_mss,speed_ms,0,blend_radius_m)
    |   movel([0.105187, -1.288026, -2.579851, -0.844512, 1.570796, 1.675984],accel_mss,speed_ms,0,blend_radius_m)
    |   movel([0.103865, -1.290394, -2.578427, -0.843568, 1.570796, 1.674661],accel_mss,speed_ms,0,blend_radius_m)
    |   movel([0.102549, -1.292754, -2.577001, -0.842634, 1.570796, 1.673345],accel_mss,speed_ms,0,blend_radius_m)
    |   speed_ms = 0.005
    |   # Splitting Linear movement in 6 (instruction 514: MoveL 436)
    |   movel([0.102549, -1.294110, -2.577744, -0.840536, 1.570796, 1.673345],accel_mss,speed_ms,0,blend_radius_m)
    |   movel([0.102549, -1.295470, -2.578485, -0.838434, 1.570796, 1.673345],accel_mss,speed_ms,0,blend_radius_m)
    |   movel([0.102549, -1.296836, -2.579225, -0.836329, 1.570796, 1.673345],accel_mss,speed_ms,0,blend_radius_m)
    |   movel([0.102549, -1.298206, -2.579963, -0.834220, 1.570796, 1.673345],accel_mss,speed_ms,0,blend_radius_m)
    |   movel([0.102549, -1.299581, -2.580699, -0.832108, 1.570796, 1.673345],accel_mss,speed_ms,0,blend_radius_m)
    |   movel([0.102549, -1.300961, -2.581435, -0.829993, 1.570796, 1.673345],accel_mss,speed_ms,0,blend_radius_m)
    |   speed_ms = 0.035
    |   # Splitting Linear movement in 6 (instruction 516: MoveL 437)
    |   movel([0.104345, -1.300434, -2.581758, -0.830198, 1.570796, 1.675142],accel_mss,speed_ms,0,blend_radius_m)
